LIN {X 0,Y 586.31,Z 664.399,A -85,B 0,C 180,E1 -9232.595,E2 -9232.595} C_VEL
LIN {X 0,Y 580.934,Z 684.929,A -85,B 0,C 180,E1 -9232.486,E2 -9232.486} C_VEL
LIN {X 0,Y 580.191,Z 691.532,A -85,B 0,C 180,E1 -9232.53,E2 -9232.53} C_VEL
LIN {X 0,Y 578.713,Z 743.986,A -85,B 0,C 180,E1 -9233.273,E2 -9233.273} C_VEL
LIN {X 0,Y 577.312,Z 767.92,A -85,B 0,C 180,E1 -9233.781,E2 -9233.781} C_VEL
LIN {X 0,Y 575.729,Z 789.042,A -85,B 0,C 180,E1 -9234.367,E2 -9234.367} C_VEL
LIN {X 0,Y 573.476,Z 813.615,A -85,B 0,C 180,E1 -9235.24,E2 -9235.24} C_VEL
LIN {X 0,Y 571.275,Z 833.863,A -85,B 0,C 180,E1 -9236.12,E2 -9236.12} C_VEL
LIN {X 0,Y 568.599,Z 856.085,A -85,B 0,C 180,E1 -9237.266,E2 -9237.266} C_VEL
LIN {X 0,Y 565.934,Z 875.723,A -85,B 0,C 180,E1 -9238.468,E2 -9238.468} C_VEL
LIN {X 0,Y 562.986,Z 896.638,A -85,B 0,C 180,E1 -9239.944,E2 -9239.944} C_VEL
LIN {X 0,Y 560.079,Z 915.772,A -85,B 0,C 180,E1 -9241.532,E2 -9241.532} C_VEL
LIN {X 0,Y 557.469,Z 932.739,A -85,B 0,C 180,E1 -9243.128,E2 -9243.128} C_VEL
LIN {X 0,Y 554.693,Z 950.508,A -85,B 0,C 180,E1 -9245.055,E2 -9245.055} C_VEL
LIN {X 0,Y 552.453,Z 965.214,A -85,B 0,C 180,E1 -9246.874,E2 -9246.874} C_VEL
LIN {X 0,Y 550.12,Z 981.104,A -85,B 0,C 180,E1 -9249.13,E2 -9249.13} C_VEL
LIN {X 0,Y 548.462,Z 993.237,A -85,B 0,C 180,E1 -9251.118,E2 -9251.118} C_VEL
LIN {X 0,Y 546.884,Z 1006.084,A -85,B 0,C 180,E1 -9253.537,E2 -9253.537} C_VEL
LIN {X 0,Y 545.776,Z 1016.202,A -85,B 0,C 180,E1 -9255.789,E2 -9255.789} C_VEL
LIN {X 0,Y 544.95,Z 1025.658,A -85,B 0,C 180,E1 -9258.249,E2 -9258.249} C_VEL
LIN {X 0,Y 544.408,Z 1033.231,A -85,B 0,C 180,E1 -9260.699,E2 -9260.699} C_VEL
LIN {X 0,Y 544.119,Z 1039.11,A -85,B 0,C 180,E1 -9263.034,E2 -9263.034} C_VEL
LIN {X 0,Y 543.975,Z 1043.859,A -85,B 0,C 180,E1 -9265.572,E2 -9265.572} C_VEL
LIN {X 0,Y 543.935,Z 1046.719,A -85,B 0,C 180,E1 -9267.788,E2 -9267.788} C_VEL
LIN {X 0,Y 543.91,Z 1048.63,A -85,B 0,C 180,E1 -9270.316,E2 -9270.316} C_VEL
LIN {X 0,Y 543.904,Z 1048.85,A -85,B 0,C 180,E1 -9272.74,E2 -9272.74} C_VEL
LIN {X 0,Y 543.911,Z 1047.945,A -85,B 0,C 180,E1 -9274.875,E2 -9274.875} C_VEL
LIN {X 0,Y 543.943,Z 1045.533,A -85,B 0,C 180,E1 -9277.393,E2 -9277.393} C_VEL
LIN {X 0,Y 544.029,Z 1041.559,A -85,B 0,C 180,E1 -9279.842,E2 -9279.842} C_VEL
LIN {X 0,Y 544.229,Z 1036.691,A -85,B 0,C 180,E1 -9282.09,E2 -9282.09} C_VEL
LIN {X 0,Y 544.667,Z 1029.45,A -85,B 0,C 180,E1 -9284.675,E2 -9284.675} C_VEL
LIN {X 0,Y 545.249,Z 1021.983,A -85,B 0,C 180,E1 -9286.843,E2 -9286.843} C_VEL
LIN {X 0,Y 546.21,Z 1012.263,A -85,B 0,C 180,E1 -9289.239,E2 -9289.239} C_VEL
LIN {X 0,Y 547.47,Z 1001.093,A -85,B 0,C 180,E1 -9291.537,E2 -9291.537} C_VEL
LIN {X 0,Y 549.156,Z 988.247,A -85,B 0,C 180,E1 -9293.842,E2 -9293.842} C_VEL
LIN {X 0,Y 551.198,Z 973.856,A -85,B 0,C 180,E1 -9296.04,E2 -9296.04} C_VEL
LIN {X 0,Y 553.43,Z 959.175,A -85,B 0,C 180,E1 -9298.018,E2 -9298.018} C_VEL
LIN {X 0,Y 556.081,Z 942.25,A -85,B 0,C 180,E1 -9299.992,E2 -9299.992} C_VEL
LIN {X 0,Y 558.6,Z 926.284,A -85,B 0,C 180,E1 -9301.632,E2 -9301.632} C_VEL
LIN {X 0,Y 561.851,Z 905.525,A -85,B 0,C 180,E1 -9303.483,E2 -9303.483} C_VEL
LIN {X 0,Y 564.509,Z 887.997,A -85,B 0,C 180,E1 -9304.836,E2 -9304.836} C_VEL
LIN {X 0,Y 567.634,Z 866.271,A -85,B 0,C 180,E1 -9306.289,E2 -9306.289} C_VEL
LIN {X 0,Y 570.163,Z 846.787,A -85,B 0,C 180,E1 -9307.399,E2 -9307.399} C_VEL
LIN {X 0,Y 572.736,Z 825.719,A -85,B 0,C 180,E1 -9308.426,E2 -9308.426} C_VEL
LIN {X 0,Y 575.102,Z 802.41,A -85,B 0,C 180,E1 -9309.358,E2 -9309.358} C_VEL
LIN {X 0,Y 577.063,Z 780.294,A -85,B 0,C 180,E1 -9310.073,E2 -9310.073} C_VEL
LIN {X 0,Y 578.78,Z 755.543,A -85,B 0,C 180,E1 -9310.679,E2 -9310.679} C_VEL
LIN {X 0,Y 579.816,Z 733.707,A -85,B 0,C 180,E1 -9311.068,E2 -9311.068} C_VEL
LIN {X 0,Y 586.618,Z 484.146,A -85,B 0,C 180,E1 -9314.52,E2 -9314.52} C_VEL
LIN {X 0,Y 588.402,Z 417.526,A -85,B 0,C 180,E1 -9315.46,E2 -9315.46} C_VEL
LIN {X 0,Y 575.019,Z 395.806,A -85,B 0,C 180,E1 -9317.164,E2 -9317.164} C_VEL
LIN {X 0,Y 561.085,Z 375.029,A -85,B 0,C 180,E1 -9319.053,E2 -9319.053} C_VEL
LIN {X 0,Y 553.737,Z 365.162,A -85,B 0,C 180,E1 -9320.097,E2 -9320.097} C_VEL
LIN {X 0,Y 550.099,Z 360.585,A -85,B 0,C 180,E1 -9320.627,E2 -9320.627} C_VEL
LIN {X 0,Y 549.271,Z 359.092,A -85,B 0,C 180,E1 -9320.758,E2 -9320.758} C_VEL
LIN {X 0,Y 546.699,Z 356.549,A -85,B 0,C 180,E1 -9321.129,E2 -9321.129} C_VEL
LIN {X 0,Y 545.557,Z 353.379,A -85,B 0,C 180,E1 -9321.337,E2 -9321.337} C_VEL
LIN {X 0,Y 545.5,Z 353.228,A -85,B 0,C 180,E1 -9324.654,E2 -9324.654} C_VEL
LIN {X 0,Y 545.56,Z 353.263,A -85,B 0,C 180,E1 -9327.893,E2 -9327.893} C_VEL
LIN {X 0,Y 545.51,Z 353.27,A -85,B 0,C 180,E1 -9331.06,E2 -9331.06} C_VEL
LIN {X 0,Y 545.517,Z 353.264,A -85,B 0,C 180,E1 -9334.486,E2 -9334.486} C_VEL
LIN {X 0,Y 545.558,Z 353.262,A -85,B 0,C 180,E1 -9337.752,E2 -9337.752} C_VEL
LIN {X 0,Y 545.507,Z 353.276,A -85,B 0,C 180,E1 -9341.051,E2 -9341.051} C_VEL
LIN {X 0,Y 545.541,Z 353.274,A -85,B 0,C 180,E1 -9344.37,E2 -9344.37} C_VEL
LIN {X 0,Y 545.517,Z 353.274,A -85,B 0,C 180,E1 -9347.509,E2 -9347.509} C_VEL
LIN {X 0,Y 545.506,Z 353.269,A -85,B 0,C 180,E1 -9350.93,E2 -9350.93} C_VEL
LIN {X 0,Y 545.561,Z 353.256,A -85,B 0,C 180,E1 -9354.109,E2 -9354.109} C_VEL
LIN {X 0,Y 545.504,Z 353.277,A -85,B 0,C 180,E1 -9357.394,E2 -9357.394} C_VEL
LIN {X 0,Y 545.533,Z 353.276,A -85,B 0,C 180,E1 -9360.735,E2 -9360.735} C_VEL
LIN {X 0,Y 545.532,Z 353.266,A -85,B 0,C 180,E1 -9363.994,E2 -9363.994} C_VEL
LIN {X 0,Y 545.502,Z 353.258,A -85,B 0,C 180,E1 -9367.266,E2 -9367.266} C_VEL
LIN {X 0,Y 545.559,Z 353.259,A -85,B 0,C 180,E1 -9370.454,E2 -9370.454} C_VEL
LIN {X 0,Y 545.504,Z 353.279,A -85,B 0,C 180,E1 -9373.719,E2 -9373.719} C_VEL
LIN {X 0,Y 545.528,Z 353.275,A -85,B 0,C 180,E1 -9377.053,E2 -9377.053} C_VEL
LIN {X 0,Y 545.531,Z 353.26,A -85,B 0,C 180,E1 -9380.268,E2 -9380.268} C_VEL
LIN {X 0,Y 545.502,Z 353.26,A -85,B 0,C 180,E1 -9383.553,E2 -9383.553} C_VEL
LIN {X 0,Y 545.562,Z 353.256,A -85,B 0,C 180,E1 -9386.803,E2 -9386.803} C_VEL
LIN {X 0,Y 545.503,Z 353.277,A -85,B 0,C 180,E1 -9389.905,E2 -9389.905} C_VEL
LIN {X 0,Y 545.538,Z 353.275,A -85,B 0,C 180,E1 -9393.232,E2 -9393.232} C_VEL
LIN {X 0,Y 545.522,Z 353.277,A -85,B 0,C 180,E1 -9396.432,E2 -9396.432} C_VEL
LIN {X 0,Y 545.547,Z 353.434,A -85,B 0,C 180,E1 -9398.499,E2 -9398.499} C_VEL
LIN {X 0,Y 546.943,Z 356.866,A -85,B 0,C 180,E1 -9399.103,E2 -9399.103} C_VEL
LIN {X 0,Y 552.731,Z 369.791,A -85,B 0,C 180,E1 -9401.346,E2 -9401.346} C_VEL
LIN {X 0,Y 553.923,Z 372.421,A -85,B 0,C 180,E1 -9401.731,E2 -9401.731} C_VEL
LIN {X 0,Y 566.29,Z 390.72,A -85,B 0,C 180,E1 -9403.483,E2 -9403.483} C_VEL
LIN {X 0,Y 578.478,Z 410.325,A -85,B 0,C 180,E1 -9405.11,E2 -9405.11} C_VEL
LIN {X 0,Y 588.478,Z 427.51,A -85,B 0,C 180,E1 -9406.38,E2 -9406.38} C_VEL
LIN {X 0,Y 581.411,Z 686.07,A -85,B 0,C 180,E1 -9409.961,E2 -9409.961} C_VEL
LIN {X 0,Y 579.185,Z 765.672,A -85,B 0,C 180,E1 -9411.076,E2 -9411.076} C_VEL
LIN {X 0,Y 577.58,Z 791.315,A -85,B 0,C 180,E1 -9411.595,E2 -9411.595} C_VEL
LIN {X 0,Y 575.8,Z 813.335,A -85,B 0,C 180,E1 -9412.197,E2 -9412.197} C_VEL
LIN {X 0,Y 573.376,Z 838.25,A -85,B 0,C 180,E1 -9413.076,E2 -9413.076} C_VEL
LIN {X 0,Y 571.195,Z 857.607,A -85,B 0,C 180,E1 -9413.91,E2 -9413.91} C_VEL
LIN {X 0,Y 568.389,Z 880.253,A -85,B 0,C 180,E1 -9415.062,E2 -9415.062} C_VEL
LIN {X 0,Y 565.532,Z 900.948,A -85,B 0,C 180,E1 -9416.322,E2 -9416.322} C_VEL
LIN {X 0,Y 562.652,Z 920.988,A -85,B 0,C 180,E1 -9417.723,E2 -9417.723} C_VEL
LIN {X 0,Y 559.666,Z 940.68,A -85,B 0,C 180,E1 -9419.332,E2 -9419.332} C_VEL
LIN {X 0,Y 557.039,Z 958.054,A -85,B 0,C 180,E1 -9420.947,E2 -9420.947} C_VEL
LIN {X 0,Y 554.171,Z 976.838,A -85,B 0,C 180,E1 -9422.955,E2 -9422.955} C_VEL
LIN {X 0,Y 551.96,Z 991.974,A -85,B 0,C 180,E1 -9424.804,E2 -9424.804} C_VEL
LIN {X 0,Y 549.686,Z 1008.315,A -85,B 0,C 180,E1 -9427.091,E2 -9427.091} C_VEL
LIN {X 0,Y 548.05,Z 1021.164,A -85,B 0,C 180,E1 -9429.159,E2 -9429.159} C_VEL
LIN {X 0,Y 546.494,Z 1034.945,A -85,B 0,C 180,E1 -9431.73,E2 -9431.73} C_VEL
LIN {X 0,Y 545.565,Z 1044.534,A -85,B 0,C 180,E1 -9433.825,E2 -9433.825} C_VEL
LIN {X 0,Y 544.805,Z 1054.257,A -85,B 0,C 180,E1 -9436.305,E2 -9436.305} C_VEL
LIN {X 0,Y 544.338,Z 1061.76,A -85,B 0,C 180,E1 -9438.665,E2 -9438.665} C_VEL
LIN {X 0,Y 544.07,Z 1067.856,A -85,B 0,C 180,E1 -9441.013,E2 -9441.013} C_VEL
LIN {X 0,Y 543.949,Z 1072.766,A -85,B 0,C 180,E1 -9443.562,E2 -9443.562} C_VEL
LIN {X 0,Y 543.918,Z 1075.604,A -85,B 0,C 180,E1 -9445.677,E2 -9445.677} C_VEL
LIN {X 0,Y 543.91,Z 1077.486,A -85,B 0,C 180,E1 -9447.998,E2 -9447.998} C_VEL
LIN {X 0,Y 543.902,Z 1077.918,A -85,B 0,C 180,E1 -9450.527,E2 -9450.527} C_VEL
LIN {X 0,Y 543.912,Z 1077.003,A -85,B 0,C 180,E1 -9452.74,E2 -9452.74} C_VEL
LIN {X 0,Y 543.934,Z 1074.679,A -85,B 0,C 180,E1 -9455.168,E2 -9455.168} C_VEL
LIN {X 0,Y 543.986,Z 1070.71,A -85,B 0,C 180,E1 -9457.605,E2 -9457.605} C_VEL
LIN {X 0,Y 544.145,Z 1066.055,A -85,B 0,C 180,E1 -9459.733,E2 -9459.733} C_VEL
LIN {X 0,Y 544.484,Z 1059.287,A -85,B 0,C 180,E1 -9462.192,E2 -9462.192} C_VEL
LIN {X 0,Y 545.031,Z 1051.054,A -85,B 0,C 180,E1 -9464.556,E2 -9464.556} C_VEL
LIN {X 0,Y 545.787,Z 1042.23,A -85,B 0,C 180,E1 -9466.716,E2 -9466.716} C_VEL
LIN {X 0,Y 547.007,Z 1030.206,A -85,B 0,C 180,E1 -9469.21,E2 -9469.21} C_VEL
LIN {X 0,Y 548.367,Z 1018.548,A -85,B 0,C 180,E1 -9471.289,E2 -9471.289} C_VEL
LIN {X 0,Y 550.294,Z 1003.93,A -85,B 0,C 180,E1 -9473.562,E2 -9473.562} C_VEL
LIN {X 0,Y 552.309,Z 989.361,A -85,B 0,C 180,E1 -9475.523,E2 -9475.523} C_VEL
LIN {X 0,Y 554.838,Z 972.333,A -85,B 0,C 180,E1 -9477.544,E2 -9477.544} C_VEL
LIN {X 0,Y 557.462,Z 954.481,A -85,B 0,C 180,E1 -9479.372,E2 -9479.372} C_VEL
LIN {X 0,Y 560.362,Z 935.264,A -85,B 0,C 180,E1 -9481.103,E2 -9481.103} C_VEL
LIN {X 0,Y 563.173,Z 915.778,A -85,B 0,C 180,E1 -9482.605,E2 -9482.605} C_VEL
LIN {X 0,Y 565.83,Z 896.882,A -85,B 0,C 180,E1 -9483.885,E2 -9483.885} C_VEL
LIN {X 0,Y 568.774,Z 873.901,A -85,B 0,C 180,E1 -9485.213,E2 -9485.213} C_VEL
LIN {X 0,Y 571.274,Z 853.014,A -85,B 0,C 180,E1 -9486.23,E2 -9486.23} C_VEL
LIN {X 0,Y 573.845,Z 828.285,A -85,B 0,C 180,E1 -9487.222,E2 -9487.222} C_VEL
LIN {X 0,Y 575.738,Z 807.183,A -85,B 0,C 180,E1 -9487.902,E2 -9487.902} C_VEL
LIN {X 0,Y 577.644,Z 781.289,A -85,B 0,C 180,E1 -9488.542,E2 -9488.542} C_VEL
LIN {X 0,Y 578.728,Z 759.201,A -85,B 0,C 180,E1 -9488.935,E2 -9488.935} C_VEL
LIN {X 0,Y 584.808,Z 519.513,A -85,B 0,C 180,E1 -9492.223,E2 -9492.223} C_VEL
LIN {X 0,Y 587.154,Z 426.916,A -85,B 0,C 180,E1 -9493.511,E2 -9493.511} C_VEL
LIN {X 0,Y 571.809,Z 400.651,A -85,B 0,C 180,E1 -9495.388,E2 -9495.388} C_VEL
LIN {X 0,Y 559.047,Z 380.64,A -85,B 0,C 180,E1 -9497.043,E2 -9497.043} C_VEL
LIN {X 0,Y 553.395,Z 371.842,A -85,B 0,C 180,E1 -9497.837,E2 -9497.837} C_VEL
LIN {X 0,Y 548.431,Z 360.447,A -85,B 0,C 180,E1 -9499.667,E2 -9499.667} C_VEL
LIN {X 0,Y 545.613,Z 353.686,A -85,B 0,C 180,E1 -9500.784,E2 -9500.784} C_VEL
LIN {X 0,Y 545.563,Z 353.268,A -85,B 0,C 180,E1 -9500.915,E2 -9500.915} C_VEL
LIN {X 0,Y 545.503,Z 353.282,A -85,B 0,C 180,E1 -9504.217,E2 -9504.217} C_VEL
LIN {X 0,Y 545.533,Z 353.276,A -85,B 0,C 180,E1 -9507.518,E2 -9507.518} C_VEL
LIN {X 0,Y 545.517,Z 353.275,A -85,B 0,C 180,E1 -9510.579,E2 -9510.579} C_VEL
LIN {X 0,Y 545.507,Z 353.274,A -85,B 0,C 180,E1 -9514.019,E2 -9514.019} C_VEL
LIN {X 0,Y 545.567,Z 353.251,A -85,B 0,C 180,E1 -9517.25,E2 -9517.25} C_VEL
LIN {X 0,Y 545.502,Z 353.261,A -85,B 0,C 180,E1 -9520.512,E2 -9520.512} C_VEL
LIN {X 0,Y 545.531,Z 353.274,A -85,B 0,C 180,E1 -9523.827,E2 -9523.827} C_VEL
LIN {X 0,Y 545.522,Z 353.268,A -85,B 0,C 180,E1 -9526.971,E2 -9526.971} C_VEL
LIN {X 0,Y 545.505,Z 353.253,A -85,B 0,C 180,E1 -9530.292,E2 -9530.292} C_VEL
LIN {X 0,Y 545.571,Z 353.272,A -85,B 0,C 180,E1 -9533.581,E2 -9533.581} C_VEL
LIN {X 0,Y 545.505,Z 353.27,A -85,B 0,C 180,E1 -9536.848,E2 -9536.848} C_VEL
LIN {X 0,Y 545.521,Z 353.252,A -85,B 0,C 180,E1 -9540.21,E2 -9540.21} C_VEL
LIN {X 0,Y 545.534,Z 353.275,A -85,B 0,C 180,E1 -9543.362,E2 -9543.362} C_VEL
LIN {X 0,Y 545.504,Z 353.259,A -85,B 0,C 180,E1 -9546.631,E2 -9546.631} C_VEL
LIN {X 0,Y 545.561,Z 353.262,A -85,B 0,C 180,E1 -9549.814,E2 -9549.814} C_VEL
LIN {X 0,Y 545.509,Z 353.276,A -85,B 0,C 180,E1 -9553.137,E2 -9553.137} C_VEL
LIN {X 0,Y 545.519,Z 353.257,A -85,B 0,C 180,E1 -9556.541,E2 -9556.541} C_VEL
LIN {X 0,Y 545.545,Z 353.267,A -85,B 0,C 180,E1 -9559.709,E2 -9559.709} C_VEL
LIN {X 0,Y 545.508,Z 353.279,A -85,B 0,C 180,E1 -9562.981,E2 -9562.981} C_VEL
LIN {X 0,Y 545.562,Z 353.255,A -85,B 0,C 180,E1 -9566.212,E2 -9566.212} C_VEL
LIN {X 0,Y 545.51,Z 353.258,A -85,B 0,C 180,E1 -9569.422,E2 -9569.422} C_VEL
LIN {X 0,Y 545.518,Z 353.261,A -85,B 0,C 180,E1 -9572.857,E2 -9572.857} C_VEL
LIN {X 0,Y 545.552,Z 353.265,A -85,B 0,C 180,E1 -9576.073,E2 -9576.073} C_VEL
LIN {X 0,Y 545.505,Z 353.271,A -85,B 0,C 180,E1 -9579.361,E2 -9579.361} C_VEL
LIN {X 0,Y 545.556,Z 353.244,A -85,B 0,C 180,E1 -9582.555,E2 -9582.555} C_VEL
LIN {X 0,Y 545.524,Z 353.391,A -85,B 0,C 180,E1 -9583.36,E2 -9583.36} C_VEL
LIN {X 0,Y 546.695,Z 356.539,A -85,B 0,C 180,E1 -9583.556,E2 -9583.556} C_VEL
LIN {X 0,Y 549.535,Z 359.67,A -85,B 0,C 180,E1 -9583.941,E2 -9583.941} C_VEL
LIN {X 0,Y 552.166,Z 363.52,A -85,B 0,C 180,E1 -9584.31,E2 -9584.31} C_VEL
LIN {X 0,Y 562.945,Z 378.525,A -85,B 0,C 180,E1 -9585.746,E2 -9585.746} C_VEL
LIN {X 0,Y 577.16,Z 400.506,A -85,B 0,C 180,E1 -9587.545,E2 -9587.545} C_VEL
LIN {X 0,Y 587.285,Z 417.698,A -85,B 0,C 180,E1 -9588.768,E2 -9588.768} C_VEL
LIN {X 0,Y 580.842,Z 665.424,A -85,B 0,C 180,E1 -9592.174,E2 -9592.174} C_VEL
LIN {X 0,Y 580.191,Z 691.532,A -85,B 0,C 180,E1 -9592.53,E2 -9592.53} C_VEL
LIN {X 0,Y 579.237,Z 699.223,A -85,B 0,C 180,E1 -9592.574,E2 -9592.574} C_VEL
LIN {X 0,Y 573.858,Z 719.75,A -85,B 0,C 180,E1 -9592.463,E2 -9592.463} C_VEL
LIN {X 0,Y 573.08,Z 726.354,A -85,B 0,C 180,E1 -9592.505,E2 -9592.505} C_VEL
LIN {X 0,Y 572.003,Z 751.824,A -85,B 0,C 180,E1 -9592.929,E2 -9592.929} C_VEL
LIN {X 0,Y 570.686,Z 772.366,A -85,B 0,C 180,E1 -9593.398,E2 -9593.398} C_VEL
LIN {X 0,Y 568.636,Z 797.064,A -85,B 0,C 180,E1 -9594.137,E2 -9594.137} C_VEL
LIN {X 0,Y 566.572,Z 817.66,A -85,B 0,C 180,E1 -9594.917,E2 -9594.917} C_VEL
LIN {X 0,Y 564.003,Z 840.035,A -85,B 0,C 180,E1 -9595.929,E2 -9595.929} C_VEL
LIN {X 0,Y 561.11,Z 861.963,A -85,B 0,C 180,E1 -9597.138,E2 -9597.138} C_VEL
LIN {X 0,Y 558.208,Z 882.64,A -85,B 0,C 180,E1 -9598.463,E2 -9598.463} C_VEL
LIN {X 0,Y 555.065,Z 903.039,A -85,B 0,C 180,E1 -9600.008,E2 -9600.008} C_VEL
LIN {X 0,Y 552.221,Z 921.02,A -85,B 0,C 180,E1 -9601.562,E2 -9601.562} C_VEL
LIN {X 0,Y 549.207,Z 939.328,A -85,B 0,C 180,E1 -9603.393,E2 -9603.393} C_VEL
LIN {X 0,Y 546.755,Z 954.528,A -85,B 0,C 180,E1 -9605.126,E2 -9605.126} C_VEL
LIN {X 0,Y 543.979,Z 971.939,A -85,B 0,C 180,E1 -9607.408,E2 -9607.408} C_VEL
LIN {X 0,Y 542.016,Z 984.923,A -85,B 0,C 180,E1 -9609.369,E2 -9609.369} C_VEL
LIN {X 0,Y 539.993,Z 999.294,A -85,B 0,C 180,E1 -9611.876,E2 -9611.876} C_VEL
LIN {X 0,Y 538.655,Z 1010.001,A -85,B 0,C 180,E1 -9614.061,E2 -9614.061} C_VEL
LIN {X 0,Y 537.499,Z 1020.862,A -85,B 0,C 180,E1 -9616.663,E2 -9616.663} C_VEL
LIN {X 0,Y 536.808,Z 1028.736,A -85,B 0,C 180,E1 -9618.939,E2 -9618.939} C_VEL
LIN {X 0,Y 536.338,Z 1035.901,A -85,B 0,C 180,E1 -9621.423,E2 -9621.423} C_VEL
LIN {X 0,Y 536.068,Z 1041.325,A -85,B 0,C 180,E1 -9623.897,E2 -9623.897} C_VEL
LIN {X 0,Y 535.965,Z 1045.057,A -85,B 0,C 180,E1 -9626.149,E2 -9626.149} C_VEL
LIN {X 0,Y 535.926,Z 1047.938,A -85,B 0,C 180,E1 -9628.824,E2 -9628.824} C_VEL
LIN {X 0,Y 535.915,Z 1049.006,A -85,B 0,C 180,E1 -9631.069,E2 -9631.069} C_VEL
LIN {X 0,Y 535.915,Z 1048.946,A -85,B 0,C 180,E1 -9633.316,E2 -9633.316} C_VEL
LIN {X 0,Y 535.937,Z 1047.259,A -85,B 0,C 180,E1 -9636.057,E2 -9636.057} C_VEL
LIN {X 0,Y 535.982,Z 1044.441,A -85,B 0,C 180,E1 -9638.367,E2 -9638.367} C_VEL
LIN {X 0,Y 536.119,Z 1040.085,A -85,B 0,C 180,E1 -9640.858,E2 -9640.858} C_VEL
LIN {X 0,Y 536.43,Z 1034.004,A -85,B 0,C 180,E1 -9643.364,E2 -9643.364} C_VEL
LIN {X 0,Y 536.937,Z 1027.114,A -85,B 0,C 180,E1 -9645.665,E2 -9645.665} C_VEL
LIN {X 0,Y 537.836,Z 1017.399,A -85,B 0,C 180,E1 -9648.312,E2 -9648.312} C_VEL
LIN {X 0,Y 538.943,Z 1007.721,A -85,B 0,C 180,E1 -9650.527,E2 -9650.527} C_VEL
LIN {X 0,Y 540.651,Z 994.638,A -85,B 0,C 180,E1 -9653.084,E2 -9653.084} C_VEL
LIN {X 0,Y 542.438,Z 982.245,A -85,B 0,C 180,E1 -9655.166,E2 -9655.166} C_VEL
LIN {X 0,Y 544.874,Z 966.806,A -85,B 0,C 180,E1 -9657.426,E2 -9657.426} C_VEL
LIN {X 0,Y 547.286,Z 951.914,A -85,B 0,C 180,E1 -9659.317,E2 -9659.317} C_VEL
LIN {X 0,Y 550.212,Z 934.606,A -85,B 0,C 180,E1 -9661.254,E2 -9661.254} C_VEL
LIN {X 0,Y 553.189,Z 916.48,A -85,B 0,C 180,E1 -9662.998,E2 -9662.998} C_VEL
LIN {X 0,Y 556.389,Z 896.896,A -85,B 0,C 180,E1 -9664.654,E2 -9664.654} C_VEL
LIN {X 0,Y 559.532,Z 876.209,A -85,B 0,C 180,E1 -9666.137,E2 -9666.137} C_VEL
LIN {X 0,Y 562.581,Z 855.295,A -85,B 0,C 180,E1 -9667.434,E2 -9667.434} C_VEL
LIN {X 0,Y 565.399,Z 833.348,A -85,B 0,C 180,E1 -9668.57,E2 -9668.57} C_VEL
LIN {X 0,Y 567.648,Z 814.001,A -85,B 0,C 180,E1 -9669.421,E2 -9669.421} C_VEL
LIN {X 0,Y 570.061,Z 789.555,A -85,B 0,C 180,E1 -9670.301,E2 -9670.301} C_VEL
LIN {X 0,Y 571.773,Z 768.263,A -85,B 0,C 180,E1 -9670.9,E2 -9670.9} C_VEL
LIN {X 0,Y 573.277,Z 744.413,A -85,B 0,C 180,E1 -9671.413,E2 -9671.413} C_VEL
LIN {X 0,Y 574.895,Z 692.081,A -85,B 0,C 180,E1 -9672.167,E2 -9672.167} C_VEL
LIN {X 0,Y 582.054,Z 442.595,A -85,B 0,C 180,E1 -9675.648,E2 -9675.648} C_VEL
LIN {X 0,Y 582.588,Z 420.937,A -85,B 0,C 180,E1 -9675.965,E2 -9675.965} C_VEL
LIN {X 0,Y 570.546,Z 401.354,A -85,B 0,C 180,E1 -9677.533,E2 -9677.533} C_VEL
LIN {X 0,Y 557.188,Z 381.281,A -85,B 0,C 180,E1 -9679.382,E2 -9679.382} C_VEL
LIN {X 0,Y 548.562,Z 369.951,A -85,B 0,C 180,E1 -9680.63,E2 -9680.63} C_VEL
LIN {X 0,Y 545.139,Z 365.328,A -85,B 0,C 180,E1 -9681.149,E2 -9681.149} C_VEL
LIN {X 0,Y 542.298,Z 361.709,A -85,B 0,C 180,E1 -9681.584,E2 -9681.584} C_VEL
LIN {X 0,Y 541.197,Z 359.978,A -85,B 0,C 180,E1 -9681.762,E2 -9681.762} C_VEL
LIN {X 0,Y 538.622,Z 357.309,A -85,B 0,C 180,E1 -9682.154,E2 -9682.154} C_VEL
LIN {X 0,Y 537.573,Z 354.248,A -85,B 0,C 180,E1 -9682.371,E2 -9682.371} C_VEL
LIN {X 0,Y 537.62,Z 354.227,A -85,B 0,C 180,E1 -9685.699,E2 -9685.699} C_VEL
LIN {X 0,Y 537.569,Z 354.256,A -85,B 0,C 180,E1 -9688.987,E2 -9688.987} C_VEL
LIN {X 0,Y 537.581,Z 354.261,A -85,B 0,C 180,E1 -9692.41,E2 -9692.41} C_VEL
LIN {X 0,Y 537.617,Z 354.253,A -85,B 0,C 180,E1 -9695.73,E2 -9695.73} C_VEL
LIN {X 0,Y 537.566,Z 354.256,A -85,B 0,C 180,E1 -9699.025,E2 -9699.025} C_VEL
LIN {X 0,Y 537.599,Z 354.249,A -85,B 0,C 180,E1 -9702.352,E2 -9702.352} C_VEL
LIN {X 0,Y 537.575,Z 354.255,A -85,B 0,C 180,E1 -9705.457,E2 -9705.457} C_VEL
LIN {X 0,Y 537.571,Z 354.263,A -85,B 0,C 180,E1 -9708.846,E2 -9708.846} C_VEL
LIN {X 0,Y 537.632,Z 354.263,A -85,B 0,C 180,E1 -9712.197,E2 -9712.197} C_VEL
LIN {X 0,Y 537.571,Z 354.259,A -85,B 0,C 180,E1 -9715.537,E2 -9715.537} C_VEL
LIN {X 0,Y 537.568,Z 354.251,A -85,B 0,C 180,E1 -9719.041,E2 -9719.041} C_VEL
LIN {X 0,Y 537.619,Z 354.246,A -85,B 0,C 180,E1 -9722.238,E2 -9722.238} C_VEL
LIN {X 0,Y 537.566,Z 354.269,A -85,B 0,C 180,E1 -9725.55,E2 -9725.55} C_VEL
LIN {X 0,Y 537.592,Z 354.266,A -85,B 0,C 180,E1 -9728.881,E2 -9728.881} C_VEL
LIN {X 0,Y 537.593,Z 354.248,A -85,B 0,C 180,E1 -9732.133,E2 -9732.133} C_VEL
LIN {X 0,Y 537.562,Z 354.246,A -85,B 0,C 180,E1 -9735.426,E2 -9735.426} C_VEL
LIN {X 0,Y 537.623,Z 354.245,A -85,B 0,C 180,E1 -9738.656,E2 -9738.656} C_VEL
LIN {X 0,Y 537.569,Z 354.267,A -85,B 0,C 180,E1 -9741.954,E2 -9741.954} C_VEL
LIN {X 0,Y 537.571,Z 354.267,A -85,B 0,C 180,E1 -9745.446,E2 -9745.446} C_VEL
LIN {X 0,Y 537.636,Z 354.264,A -85,B 0,C 180,E1 -9748.796,E2 -9748.796} C_VEL
LIN {X 0,Y 537.566,Z 354.269,A -85,B 0,C 180,E1 -9752.013,E2 -9752.013} C_VEL
LIN {X 0,Y 537.581,Z 354.27,A -85,B 0,C 180,E1 -9755.445,E2 -9755.445} C_VEL
LIN {X 0,Y 537.598,Z 354.432,A -85,B 0,C 180,E1 -9757.558,E2 -9757.558} C_VEL
LIN {X 0,Y 538.888,Z 357.777,A -85,B 0,C 180,E1 -9758.161,E2 -9758.161} C_VEL
LIN {X 0,Y 541.452,Z 363.112,A -85,B 0,C 180,E1 -9759.166,E2 -9759.166} C_VEL
LIN {X 0,Y 545.365,Z 371.859,A -85,B 0,C 180,E1 -9760.677,E2 -9760.677} C_VEL
LIN {X 0,Y 558.222,Z 390.685,A -85,B 0,C 180,E1 -9762.581,E2 -9762.581} C_VEL
LIN {X 0,Y 572.345,Z 413.012,A -85,B 0,C 180,E1 -9764.529,E2 -9764.529} C_VEL
LIN {X 0,Y 582.655,Z 430.956,A -85,B 0,C 180,E1 -9765.879,E2 -9765.879} C_VEL
LIN {X 0,Y 575.261,Z 689.165,A -85,B 0,C 180,E1 -9769.484,E2 -9769.484} C_VEL
LIN {X 0,Y 573.021,Z 765.526,A -85,B 0,C 180,E1 -9770.564,E2 -9770.564} C_VEL
LIN {X 0,Y 571.362,Z 791.034,A -85,B 0,C 180,E1 -9771.083,E2 -9771.083} C_VEL
LIN {X 0,Y 569.508,Z 813.006,A -85,B 0,C 180,E1 -9771.687,E2 -9771.687} C_VEL
LIN {X 0,Y 567.08,Z 837.01,A -85,B 0,C 180,E1 -9772.532,E2 -9772.532} C_VEL
LIN {X 0,Y 564.664,Z 857.615,A -85,B 0,C 180,E1 -9773.426,E2 -9773.426} C_VEL
LIN {X 0,Y 561.706,Z 880.381,A -85,B 0,C 180,E1 -9774.596,E2 -9774.596} C_VEL
LIN {X 0,Y 558.718,Z 901.112,A -85,B 0,C 180,E1 -9775.872,E2 -9775.872} C_VEL
LIN {X 0,Y 555.626,Z 921.636,A -85,B 0,C 180,E1 -9777.325,E2 -9777.325} C_VEL
LIN {X 0,Y 552.492,Z 941.178,A -85,B 0,C 180,E1 -9778.95,E2 -9778.95} C_VEL
LIN {X 0,Y 549.706,Z 958.728,A -85,B 0,C 180,E1 -9780.608,E2 -9780.608} C_VEL
LIN {X 0,Y 546.81,Z 976.686,A -85,B 0,C 180,E1 -9782.561,E2 -9782.561} C_VEL
LIN {X 0,Y 544.466,Z 991.807,A -85,B 0,C 180,E1 -9784.433,E2 -9784.433} C_VEL
LIN {X 0,Y 542.061,Z 1008.127,A -85,B 0,C 180,E1 -9786.75,E2 -9786.75} C_VEL
LIN {X 0,Y 540.311,Z 1021.029,A -85,B 0,C 180,E1 -9788.859,E2 -9788.859} C_VEL
LIN {X 0,Y 538.643,Z 1034.899,A -85,B 0,C 180,E1 -9791.492,E2 -9791.492} C_VEL
LIN {X 0,Y 537.634,Z 1044.778,A -85,B 0,C 180,E1 -9793.69,E2 -9793.69} C_VEL
LIN {X 0,Y 536.807,Z 1054.754,A -85,B 0,C 180,E1 -9796.317,E2 -9796.317} C_VEL
LIN {X 0,Y 536.35,Z 1061.849,A -85,B 0,C 180,E1 -9798.603,E2 -9798.603} C_VEL
LIN {X 0,Y 536.065,Z 1068.155,A -85,B 0,C 180,E1 -9801.094,E2 -9801.094} C_VEL
LIN {X 0,Y 535.95,Z 1072.713,A -85,B 0,C 180,E1 -9803.573,E2 -9803.573} C_VEL
LIN {X 0,Y 535.918,Z 1075.505,A -85,B 0,C 180,E1 -9805.72,E2 -9805.72} C_VEL
LIN {X 0,Y 535.906,Z 1077.409,A -85,B 0,C 180,E1 -9808.182,E2 -9808.182} C_VEL
LIN {X 0,Y 535.906,Z 1077.682,A -85,B 0,C 180,E1 -9810.641,E2 -9810.641} C_VEL
LIN {X 0,Y 535.915,Z 1076.789,A -85,B 0,C 180,E1 -9812.78,E2 -9812.78} C_VEL
LIN {X 0,Y 535.934,Z 1074.466,A -85,B 0,C 180,E1 -9815.245,E2 -9815.245} C_VEL
LIN {X 0,Y 535.99,Z 1070.496,A -85,B 0,C 180,E1 -9817.719,E2 -9817.719} C_VEL
LIN {X 0,Y 536.155,Z 1065.839,A -85,B 0,C 180,E1 -9819.879,E2 -9819.879} C_VEL
LIN {X 0,Y 536.526,Z 1058.886,A -85,B 0,C 180,E1 -9822.432,E2 -9822.432} C_VEL
LIN {X 0,Y 537.135,Z 1050.426,A -85,B 0,C 180,E1 -9824.886,E2 -9824.886} C_VEL
LIN {X 0,Y 538.052,Z 1040.616,A -85,B 0,C 180,E1 -9827.298,E2 -9827.298} C_VEL
LIN {X 0,Y 539.349,Z 1028.823,A -85,B 0,C 180,E1 -9829.719,E2 -9829.719} C_VEL
LIN {X 0,Y 540.915,Z 1016.457,A -85,B 0,C 180,E1 -9831.925,E2 -9831.925} C_VEL
LIN {X 0,Y 543.014,Z 1001.327,A -85,B 0,C 180,E1 -9834.244,E2 -9834.244} C_VEL
LIN {X 0,Y 545.091,Z 987.372,A -85,B 0,C 180,E1 -9836.119,E2 -9836.119} C_VEL
LIN {X 0,Y 547.921,Z 969.064,A -85,B 0,C 180,E1 -9838.265,E2 -9838.265} C_VEL
LIN {X 0,Y 550.435,Z 952.988,A -85,B 0,C 180,E1 -9839.91,E2 -9839.91} C_VEL
LIN {X 0,Y 553.61,Z 932.836,A -85,B 0,C 180,E1 -9841.713,E2 -9841.713} C_VEL
LIN {X 0,Y 556.371,Z 914.575,A -85,B 0,C 180,E1 -9843.125,E2 -9843.125} C_VEL
LIN {X 0,Y 559.385,Z 894.047,A -85,B 0,C 180,E1 -9844.516,E2 -9844.516} C_VEL
LIN {X 0,Y 562.224,Z 872.47,A -85,B 0,C 180,E1 -9845.748,E2 -9845.748} C_VEL
LIN {X 0,Y 564.952,Z 850.686,A -85,B 0,C 180,E1 -9846.805,E2 -9846.805} C_VEL
LIN {X 0,Y 567.425,Z 827.51,A -85,B 0,C 180,E1 -9847.727,E2 -9847.727} C_VEL
LIN {X 0,Y 569.383,Z 806.505,A -85,B 0,C 180,E1 -9848.405,E2 -9848.405} C_VEL
LIN {X 0,Y 571.327,Z 780.86,A -85,B 0,C 180,E1 -9849.041,E2 -9849.041} C_VEL
LIN {X 0,Y 572.445,Z 758.816,A -85,B 0,C 180,E1 -9849.435,E2 -9849.435} C_VEL
LIN {X 0,Y 578.832,Z 518.494,A -85,B 0,C 180,E1 -9852.761,E2 -9852.761} C_VEL
LIN {X 0,Y 581.183,Z 430.246,A -85,B 0,C 180,E1 -9853.998,E2 -9853.998} C_VEL
LIN {X 0,Y 567.071,Z 405.931,A -85,B 0,C 180,E1 -9855.766,E2 -9855.766} C_VEL
LIN {X 0,Y 554.721,Z 386.396,A -85,B 0,C 180,E1 -9857.402,E2 -9857.402} C_VEL
LIN {X 0,Y 546.313,Z 373.784,A -85,B 0,C 180,E1 -9858.575,E2 -9858.575} C_VEL
LIN {X 0,Y 544.919,Z 371.558,A -85,B 0,C 180,E1 -9858.796,E2 -9858.796} C_VEL
LIN {X 0,Y 540.498,Z 361.439,A -85,B 0,C 180,E1 -9860.482,E2 -9860.482} C_VEL
LIN {X 0,Y 538.801,Z 357.546,A -85,B 0,C 180,E1 -9861.152,E2 -9861.152} C_VEL
LIN {X 0,Y 537.572,Z 354.265,A -85,B 0,C 180,E1 -9861.729,E2 -9861.729} C_VEL
LIN {X 0,Y 537.62,Z 354.251,A -85,B 0,C 180,E1 -9865.052,E2 -9865.052} C_VEL
LIN {X 0,Y 537.562,Z 354.258,A -85,B 0,C 180,E1 -9868.238,E2 -9868.238} C_VEL
LIN {X 0,Y 537.599,Z 354.255,A -85,B 0,C 180,E1 -9871.566,E2 -9871.566} C_VEL
LIN {X 0,Y 537.588,Z 354.264,A -85,B 0,C 180,E1 -9874.79,E2 -9874.79} C_VEL
LIN {X 0,Y 537.563,Z 354.266,A -85,B 0,C 180,E1 -9878.16,E2 -9878.16} C_VEL
LIN {X 0,Y 537.619,Z 354.241,A -85,B 0,C 180,E1 -9881.456,E2 -9881.456} C_VEL
LIN {X 0,Y 537.569,Z 354.256,A -85,B 0,C 180,E1 -9884.685,E2 -9884.685} C_VEL
LIN {X 0,Y 537.573,Z 354.267,A -85,B 0,C 180,E1 -9888.194,E2 -9888.194} C_VEL
LIN {X 0,Y 537.626,Z 354.242,A -85,B 0,C 180,E1 -9891.551,E2 -9891.551} C_VEL
LIN {X 0,Y 537.565,Z 354.251,A -85,B 0,C 180,E1 -9894.771,E2 -9894.771} C_VEL
LIN {X 0,Y 537.584,Z 354.268,A -85,B 0,C 180,E1 -9898.188,E2 -9898.188} C_VEL
LIN {X 0,Y 537.6,Z 354.237,A -85,B 0,C 180,E1 -9901.386,E2 -9901.386} C_VEL
LIN {X 0,Y 537.564,Z 354.258,A -85,B 0,C 180,E1 -9904.694,E2 -9904.694} C_VEL
LIN {X 0,Y 537.617,Z 354.259,A -85,B 0,C 180,E1 -9908.018,E2 -9908.018} C_VEL
LIN {X 0,Y 537.575,Z 354.238,A -85,B 0,C 180,E1 -9911.262,E2 -9911.262} C_VEL
LIN {X 0,Y 537.569,Z 354.259,A -85,B 0,C 180,E1 -9914.713,E2 -9914.713} C_VEL
LIN {X 0,Y 537.626,Z 354.257,A -85,B 0,C 180,E1 -9917.983,E2 -9917.983} C_VEL
LIN {X 0,Y 537.569,Z 354.245,A -85,B 0,C 180,E1 -9921.272,E2 -9921.272} C_VEL
LIN {X 0,Y 537.585,Z 354.247,A -85,B 0,C 180,E1 -9924.622,E2 -9924.622} C_VEL
LIN {X 0,Y 537.619,Z 354.263,A -85,B 0,C 180,E1 -9927.949,E2 -9927.949} C_VEL
LIN {X 0,Y 537.57,Z 354.269,A -85,B 0,C 180,E1 -9931.262,E2 -9931.262} C_VEL
LIN {X 0,Y 537.607,Z 354.258,A -85,B 0,C 180,E1 -9934.56,E2 -9934.56} C_VEL
LIN {X 0,Y 537.591,Z 354.263,A -85,B 0,C 180,E1 -9937.864,E2 -9937.864} C_VEL
LIN {X 0,Y 537.573,Z 354.271,A -85,B 0,C 180,E1 -9941.182,E2 -9941.182} C_VEL
LIN {X 0,Y 537.651,Z 354.44,A -85,B 0,C 180,E1 -9942.44,E2 -9942.44} C_VEL
LIN {X 0,Y 538.856,Z 357.626,A -85,B 0,C 180,E1 -9942.65,E2 -9942.65} C_VEL
LIN {X 0,Y 541.64,Z 360.745,A -85,B 0,C 180,E1 -9943.045,E2 -9943.045} C_VEL
LIN {X 0,Y 544.3,Z 364.596,A -85,B 0,C 180,E1 -9943.433,E2 -9943.433} C_VEL
LIN {X 0,Y 545.871,Z 366.544,A -85,B 0,C 180,E1 -9943.653,E2 -9943.653} C_VEL
LIN {X 0,Y 558.69,Z 384.425,A -85,B 0,C 180,E1 -9945.405,E2 -9945.405} C_VEL
LIN {X 0,Y 572.771,Z 406.422,A -85,B 0,C 180,E1 -9947.222,E2 -9947.222} C_VEL
LIN {X 0,Y 581.317,Z 421.073,A -85,B 0,C 180,E1 -9948.28,E2 -9948.28} C_VEL
LIN {X 0,Y 574.594,Z 667.992,A -85,B 0,C 180,E1 -9951.703,E2 -9951.703} C_VEL
LIN {X 0,Y 573.08,Z 726.354,A -85,B 0,C 180,E1 -9952.505,E2 -9952.505} C_VEL
LIN {X 0,Y 572.024,Z 734.039,A -85,B 0,C 180,E1 -9952.548,E2 -9952.548} C_VEL
LIN {X 0,Y 566.404,Z 753.361,A -85,B 0,C 180,E1 -9952.511,E2 -9952.511} C_VEL
LIN {X 0,Y 565.216,Z 760.968,A -85,B 0,C 180,E1 -9952.606,E2 -9952.606} C_VEL
LIN {X 0,Y 563.322,Z 785.096,A -85,B 0,C 180,E1 -9953.249,E2 -9953.249} C_VEL
LIN {X 0,Y 561.204,Z 807.81,A -85,B 0,C 180,E1 -9954.019,E2 -9954.019} C_VEL
LIN {X 0,Y 558.613,Z 830.665,A -85,B 0,C 180,E1 -9954.993,E2 -9954.993} C_VEL
LIN {X 0,Y 556.166,Z 849.641,A -85,B 0,C 180,E1 -9955.949,E2 -9955.949} C_VEL
LIN {X 0,Y 552.913,Z 872.771,A -85,B 0,C 180,E1 -9957.329,E2 -9957.329} C_VEL
LIN {X 0,Y 550.056,Z 891.211,A -85,B 0,C 180,E1 -9958.62,E2 -9958.62} C_VEL
LIN {X 0,Y 546.807,Z 911.299,A -85,B 0,C 180,E1 -9960.234,E2 -9960.234} C_VEL
LIN {X 0,Y 543.754,Z 929.256,A -85,B 0,C 180,E1 -9961.917,E2 -9961.917} C_VEL
LIN {X 0,Y 540.822,Z 946.72,A -85,B 0,C 180,E1 -9963.777,E2 -9963.777} C_VEL
LIN {X 0,Y 538.054,Z 962.697,A -85,B 0,C 180,E1 -9965.752,E2 -9965.752} C_VEL
LIN {X 0,Y 535.694,Z 977.225,A -85,B 0,C 180,E1 -9967.79,E2 -9967.79} C_VEL
LIN {X 0,Y 533.393,Z 991.816,A -85,B 0,C 180,E1 -9970.166,E2 -9970.166} C_VEL
LIN {X 0,Y 531.807,Z 1003.018,A -85,B 0,C 180,E1 -9972.267,E2 -9972.267} C_VEL
LIN {X 0,Y 530.282,Z 1015.096,A -85,B 0,C 180,E1 -9974.917,E2 -9974.917} C_VEL
LIN {X 0,Y 529.372,Z 1023.567,A -85,B 0,C 180,E1 -9977.122,E2 -9977.122} C_VEL
LIN {X 0,Y 528.655,Z 1032.053,A -85,B 0,C 180,E1 -9979.759,E2 -9979.759} C_VEL
LIN {X 0,Y 528.245,Z 1038.188,A -85,B 0,C 180,E1 -9982.167,E2 -9982.167} C_VEL
LIN {X 0,Y 528.036,Z 1043.216,A -85,B 0,C 180,E1 -9984.676,E2 -9984.676} C_VEL
LIN {X 0,Y 527.946,Z 1046.764,A -85,B 0,C 180,E1 -9987.286,E2 -9987.286} C_VEL
LIN {X 0,Y 527.918,Z 1048.638,A -85,B 0,C 180,E1 -9989.566,E2 -9989.566} C_VEL
LIN {X 0,Y 527.911,Z 1049.399,A -85,B 0,C 180,E1 -9992.171,E2 -9992.171} C_VEL
LIN {X 0,Y 527.915,Z 1048.551,A -85,B 0,C 180,E1 -9994.672,E2 -9994.672} C_VEL
LIN {X 0,Y 527.949,Z 1046.609,A -85,B 0,C 180,E1 -9996.962,E2 -9996.962} C_VEL
LIN {X 0,Y 528.045,Z 1042.69,A -85,B 0,C 180,E1 -9999.702,E2 -9999.702} C_VEL
LIN {X 0,Y 528.255,Z 1037.986,A -85,B 0,C 180,E1 -10002.017,E2 -10002.017} C_VEL
LIN {X 0,Y 528.707,Z 1031.428,A -85,B 0,C 180,E1 -10004.568,E2 -10004.568} C_VEL
LIN {X 0,Y 529.433,Z 1022.993,A -85,B 0,C 180,E1 -10007.135,E2 -10007.135} C_VEL
LIN {X 0,Y 530.503,Z 1013.389,A -85,B 0,C 180,E1 -10009.603,E2 -10009.603} C_VEL
LIN {X 0,Y 532.004,Z 1001.752,A -85,B 0,C 180,E1 -10012.091,E2 -10012.091} C_VEL
LIN {X 0,Y 533.792,Z 989.652,A -85,B 0,C 180,E1 -10014.337,E2 -10014.337} C_VEL
LIN {X 0,Y 536.05,Z 975.49,A -85,B 0,C 180,E1 -10016.594,E2 -10016.594} C_VEL
LIN {X 0,Y 538.508,Z 960.941,A -85,B 0,C 180,E1 -10018.623,E2 -10018.623} C_VEL
LIN {X 0,Y 541.584,Z 943.283,A -85,B 0,C 180,E1 -10020.758,E2 -10020.758} C_VEL
LIN {X 0,Y 544.361,Z 927.384,A -85,B 0,C 180,E1 -10022.436,E2 -10022.436} C_VEL
LIN {X 0,Y 547.94,Z 906.773,A -85,B 0,C 180,E1 -10024.324,E2 -10024.324} C_VEL
LIN {X 0,Y 550.833,Z 889.337,A -85,B 0,C 180,E1 -10025.704,E2 -10025.704} C_VEL
LIN {X 0,Y 554.113,Z 868.732,A -85,B 0,C 180,E1 -10027.128,E2 -10027.128} C_VEL
LIN {X 0,Y 557.021,Z 848.148,A -85,B 0,C 180,E1 -10028.33,E2 -10028.33} C_VEL
LIN {X 0,Y 559.753,Z 827.581,A -85,B 0,C 180,E1 -10029.356,E2 -10029.356} C_VEL
LIN {X 0,Y 562.402,Z 803.981,A -85,B 0,C 180,E1 -10030.327,E2 -10030.327} C_VEL
LIN {X 0,Y 564.454,Z 782.628,A -85,B 0,C 180,E1 -10031.036,E2 -10031.036} C_VEL
LIN {X 0,Y 566.444,Z 756.724,A -85,B 0,C 180,E1 -10031.692,E2 -10031.692} C_VEL
LIN {X 0,Y 567.573,Z 734.884,A -85,B 0,C 180,E1 -10032.09,E2 -10032.09} C_VEL
LIN {X 0,Y 574.974,Z 487.355,A -85,B 0,C 180,E1 -10035.575,E2 -10035.575} C_VEL
LIN {X 0,Y 576.754,Z 424.351,A -85,B 0,C 180,E1 -10036.486,E2 -10036.486} C_VEL
LIN {X 0,Y 566.099,Z 406.895,A -85,B 0,C 180,E1 -10037.909,E2 -10037.909} C_VEL
LIN {X 0,Y 553.282,Z 387.489,A -85,B 0,C 180,E1 -10039.72,E2 -10039.72} C_VEL
LIN {X 0,Y 544.456,Z 375.833,A -85,B 0,C 180,E1 -10041.023,E2 -10041.023} C_VEL
LIN {X 0,Y 541.053,Z 371.344,A -85,B 0,C 180,E1 -10041.547,E2 -10041.547} C_VEL
LIN {X 0,Y 537.278,Z 366.328,A -85,B 0,C 180,E1 -10042.144,E2 -10042.144} C_VEL
LIN {X 0,Y 534.433,Z 362.708,A -85,B 0,C 180,E1 -10042.601,E2 -10042.601} C_VEL
LIN {X 0,Y 533.576,Z 361.171,A -85,B 0,C 180,E1 -10042.75,E2 -10042.75} C_VEL
LIN {X 0,Y 530.914,Z 358.644,A -85,B 0,C 180,E1 -10043.171,E2 -10043.171} C_VEL
LIN {X 0,Y 529.721,Z 355.604,A -85,B 0,C 180,E1 -10043.404,E2 -10043.404} C_VEL
LIN {X 0,Y 529.662,Z 355.203,A -85,B 0,C 180,E1 -10043.422,E2 -10043.422} C_VEL
LIN {X 0,Y 529.628,Z 355.258,A -85,B 0,C 180,E1 -10046.756,E2 -10046.756} C_VEL
LIN {X 0,Y 529.669,Z 355.254,A -85,B 0,C 180,E1 -10050.108,E2 -10050.108} C_VEL
LIN {X 0,Y 529.646,Z 355.258,A -85,B 0,C 180,E1 -10053.301,E2 -10053.301} C_VEL
LIN {X 0,Y 529.631,Z 355.257,A -85,B 0,C 180,E1 -10056.761,E2 -10056.761} C_VEL
LIN {X 0,Y 529.686,Z 355.254,A -85,B 0,C 180,E1 -10060.064,E2 -10060.064} C_VEL
LIN {X 0,Y 529.634,Z 355.25,A -85,B 0,C 180,E1 -10063.324,E2 -10063.324} C_VEL
LIN {X 0,Y 529.631,Z 355.245,A -85,B 0,C 180,E1 -10066.795,E2 -10066.795} C_VEL
LIN {X 0,Y 529.681,Z 355.233,A -85,B 0,C 180,E1 -10070.108,E2 -10070.108} C_VEL
LIN {X 0,Y 529.627,Z 355.248,A -85,B 0,C 180,E1 -10073.387,E2 -10073.387} C_VEL
LIN {X 0,Y 529.638,Z 355.254,A -85,B 0,C 180,E1 -10076.862,E2 -10076.862} C_VEL
LIN {X 0,Y 529.69,Z 355.247,A -85,B 0,C 180,E1 -10080.216,E2 -10080.216} C_VEL
LIN {X 0,Y 529.627,Z 355.241,A -85,B 0,C 180,E1 -10083.572,E2 -10083.572} C_VEL
LIN {X 0,Y 529.634,Z 355.234,A -85,B 0,C 180,E1 -10087.049,E2 -10087.049} C_VEL
LIN {X 0,Y 529.667,Z 355.242,A -85,B 0,C 180,E1 -10090.221,E2 -10090.221} C_VEL
LIN {X 0,Y 529.625,Z 355.256,A -85,B 0,C 180,E1 -10093.539,E2 -10093.539} C_VEL
LIN {X 0,Y 529.669,Z 355.247,A -85,B 0,C 180,E1 -10096.844,E2 -10096.844} C_VEL
LIN {X 0,Y 529.64,Z 355.236,A -85,B 0,C 180,E1 -10100.096,E2 -10100.096} C_VEL
LIN {X 0,Y 529.627,Z 355.236,A -85,B 0,C 180,E1 -10103.475,E2 -10103.475} C_VEL
LIN {X 0,Y 529.683,Z 355.233,A -85,B 0,C 180,E1 -10106.762,E2 -10106.762} C_VEL
LIN {X 0,Y 529.629,Z 355.255,A -85,B 0,C 180,E1 -10110.02,E2 -10110.02} C_VEL
LIN {X 0,Y 529.64,Z 355.256,A -85,B 0,C 180,E1 -10113.454,E2 -10113.454} C_VEL
LIN {X 0,Y 529.685,Z 355.455,A -85,B 0,C 180,E1 -10116.576,E2 -10116.576} C_VEL
LIN {X 0,Y 531.295,Z 359.193,A -85,B 0,C 180,E1 -10117.301,E2 -10117.301} C_VEL
LIN {X 0,Y 536.976,Z 371.547,A -85,B 0,C 180,E1 -10119.591,E2 -10119.591} C_VEL
LIN {X 0,Y 550.839,Z 391.729,A -85,B 0,C 180,E1 -10121.739,E2 -10121.739} C_VEL
LIN {X 0,Y 562.562,Z 409.865,A -85,B 0,C 180,E1 -10123.425,E2 -10123.425} C_VEL
LIN {X 0,Y 574.643,Z 430.214,A -85,B 0,C 180,E1 -10125.069,E2 -10125.069} C_VEL
LIN {X 0,Y 576.866,Z 434.607,A -85,B 0,C 180,E1 -10125.369,E2 -10125.369} C_VEL
LIN {X 0,Y 569.179,Z 691.344,A -85,B 0,C 180,E1 -10128.984,E2 -10128.984} C_VEL
LIN {X 0,Y 566.9,Z 765.505,A -85,B 0,C 180,E1 -10130.043,E2 -10130.043} C_VEL
LIN {X 0,Y 565.176,Z 790.973,A -85,B 0,C 180,E1 -10130.566,E2 -10130.566} C_VEL
LIN {X 0,Y 563.236,Z 813.045,A -85,B 0,C 180,E1 -10131.177,E2 -10131.177} C_VEL
LIN {X 0,Y 560.692,Z 837.061,A -85,B 0,C 180,E1 -10132.03,E2 -10132.03} C_VEL
LIN {X 0,Y 558.175,Z 857.631,A -85,B 0,C 180,E1 -10132.93,E2 -10132.93} C_VEL
LIN {X 0,Y 555.075,Z 880.433,A -85,B 0,C 180,E1 -10134.115,E2 -10134.115} C_VEL
LIN {X 0,Y 552.1,Z 900.242,A -85,B 0,C 180,E1 -10135.342,E2 -10135.342} C_VEL
LIN {X 0,Y 549.066,Z 919.466,A -85,B 0,C 180,E1 -10136.707,E2 -10136.707} C_VEL
LIN {X 0,Y 545.654,Z 939.851,A -85,B 0,C 180,E1 -10138.393,E2 -10138.393} C_VEL
LIN {X 0,Y 542.725,Z 957.285,A -85,B 0,C 180,E1 -10140.048,E2 -10140.048} C_VEL
LIN {X 0,Y 539.48,Z 976.543,A -85,B 0,C 180,E1 -10142.156,E2 -10142.156} C_VEL
LIN {X 0,Y 536.998,Z 991.652,A -85,B 0,C 180,E1 -10144.051,E2 -10144.051} C_VEL
LIN {X 0,Y 534.392,Z 1008.386,A -85,B 0,C 180,E1 -10146.468,E2 -10146.468} C_VEL
LIN {X 0,Y 532.603,Z 1020.77,A -85,B 0,C 180,E1 -10148.526,E2 -10148.526} C_VEL
LIN {X 0,Y 530.883,Z 1034.172,A -85,B 0,C 180,E1 -10151.098,E2 -10151.098} C_VEL
LIN {X 0,Y 529.799,Z 1044.095,A -85,B 0,C 180,E1 -10153.329,E2 -10153.329} C_VEL
LIN {X 0,Y 528.928,Z 1053.815,A -85,B 0,C 180,E1 -10155.885,E2 -10155.885} C_VEL
LIN {X 0,Y 528.401,Z 1061.322,A -85,B 0,C 180,E1 -10158.318,E2 -10158.318} C_VEL
LIN {X 0,Y 528.114,Z 1067.163,A -85,B 0,C 180,E1 -10160.629,E2 -10160.629} C_VEL
LIN {X 0,Y 527.952,Z 1072.334,A -85,B 0,C 180,E1 -10163.366,E2 -10163.366} C_VEL
LIN {X 0,Y 527.922,Z 1075.175,A -85,B 0,C 180,E1 -10165.546,E2 -10165.546} C_VEL
LIN {X 0,Y 527.916,Z 1077.058,A -85,B 0,C 180,E1 -10167.938,E2 -10167.938} C_VEL
LIN {X 0,Y 527.908,Z 1077.492,A -85,B 0,C 180,E1 -10170.543,E2 -10170.543} C_VEL
LIN {X 0,Y 527.918,Z 1076.576,A -85,B 0,C 180,E1 -10172.823,E2 -10172.823} C_VEL
LIN {X 0,Y 527.935,Z 1074.252,A -85,B 0,C 180,E1 -10175.325,E2 -10175.325} C_VEL
LIN {X 0,Y 527.999,Z 1070.282,A -85,B 0,C 180,E1 -10177.837,E2 -10177.837} C_VEL
LIN {X 0,Y 528.179,Z 1065.365,A -85,B 0,C 180,E1 -10180.14,E2 -10180.14} C_VEL
LIN {X 0,Y 528.6,Z 1058.139,A -85,B 0,C 180,E1 -10182.786,E2 -10182.786} C_VEL
LIN {X 0,Y 529.215,Z 1050.208,A -85,B 0,C 180,E1 -10185.114,E2 -10185.114} C_VEL
LIN {X 0,Y 530.137,Z 1040.857,A -85,B 0,C 180,E1 -10187.451,E2 -10187.451} C_VEL
LIN {X 0,Y 531.499,Z 1029.162,A -85,B 0,C 180,E1 -10189.908,E2 -10189.908} C_VEL
LIN {X 0,Y 533.043,Z 1017.489,A -85,B 0,C 180,E1 -10192.034,E2 -10192.034} C_VEL
LIN {X 0,Y 535.335,Z 1001.832,A -85,B 0,C 180,E1 -10194.497,E2 -10194.497} C_VEL
LIN {X 0,Y 537.504,Z 987.941,A -85,B 0,C 180,E1 -10196.398,E2 -10196.398} C_VEL
LIN {X 0,Y 540.38,Z 970.296,A -85,B 0,C 180,E1 -10198.515,E2 -10198.515} C_VEL
LIN {X 0,Y 543.078,Z 953.791,A -85,B 0,C 180,E1 -10200.235,E2 -10200.235} C_VEL
LIN {X 0,Y 546.277,Z 934.581,A -85,B 0,C 180,E1 -10201.998,E2 -10201.998} C_VEL
LIN {X 0,Y 549.333,Z 915.171,A -85,B 0,C 180,E1 -10203.524,E2 -10203.524} C_VEL
LIN {X 0,Y 552.374,Z 895.308,A -85,B 0,C 180,E1 -10204.891,E2 -10204.891} C_VEL
LIN {X 0,Y 555.465,Z 873.063,A -85,B 0,C 180,E1 -10206.188,E2 -10206.188} C_VEL
LIN {X 0,Y 558.076,Z 853.029,A -85,B 0,C 180,E1 -10207.178,E2 -10207.178} C_VEL
LIN {X 0,Y 560.861,Z 828.542,A -85,B 0,C 180,E1 -10208.18,E2 -10208.18} C_VEL
LIN {X 0,Y 562.891,Z 807.673,A -85,B 0,C 180,E1 -10208.865,E2 -10208.865} C_VEL
LIN {X 0,Y 564.894,Z 783.094,A -85,B 0,C 180,E1 -10209.496,E2 -10209.496} C_VEL
LIN {X 0,Y 566.148,Z 759.815,A -85,B 0,C 180,E1 -10209.924,E2 -10209.924} C_VEL
LIN {X 0,Y 572.717,Z 523.949,A -85,B 0,C 180,E1 -10213.219,E2 -10213.219} C_VEL
LIN {X 0,Y 575.229,Z 433.455,A -85,B 0,C 180,E1 -10214.5,E2 -10214.5} C_VEL
LIN {X 0,Y 561.74,Z 410.227,A -85,B 0,C 180,E1 -10216.231,E2 -10216.231} C_VEL
LIN {X 0,Y 550.04,Z 391.577,A -85,B 0,C 180,E1 -10217.819,E2 -10217.819} C_VEL
LIN {X 0,Y 539.44,Z 375.609,A -85,B 0,C 180,E1 -10219.343,E2 -10219.343} C_VEL
LIN {X 0,Y 536.613,Z 371.19,A -85,B 0,C 180,E1 -10219.793,E2 -10219.793} C_VEL
LIN {X 0,Y 531.318,Z 359.259,A -85,B 0,C 180,E1 -10221.883,E2 -10221.883} C_VEL
LIN {X 0,Y 529.841,Z 356.307,A -85,B 0,C 180,E1 -10222.443,E2 -10222.443} C_VEL
LIN {X 0,Y 529.65,Z 355.241,A -85,B 0,C 180,E1 -10222.634,E2 -10222.634} C_VEL
LIN {X 0,Y 529.625,Z 355.242,A -85,B 0,C 180,E1 -10226.025,E2 -10226.025} C_VEL
LIN {X 0,Y 529.678,Z 355.232,A -85,B 0,C 180,E1 -10229.357,E2 -10229.357} C_VEL
LIN {X 0,Y 529.632,Z 355.234,A -85,B 0,C 180,E1 -10232.571,E2 -10232.571} C_VEL
LIN {X 0,Y 529.627,Z 355.237,A -85,B 0,C 180,E1 -10236.052,E2 -10236.052} C_VEL
LIN {X 0,Y 529.688,Z 355.248,A -85,B 0,C 180,E1 -10239.329,E2 -10239.329} C_VEL
LIN {X 0,Y 529.63,Z 355.253,A -85,B 0,C 180,E1 -10242.645,E2 -10242.645} C_VEL
LIN {X 0,Y 529.632,Z 355.235,A -85,B 0,C 180,E1 -10246.127,E2 -10246.127} C_VEL
LIN {X 0,Y 529.679,Z 355.235,A -85,B 0,C 180,E1 -10249.449,E2 -10249.449} C_VEL
LIN {X 0,Y 529.628,Z 355.256,A -85,B 0,C 180,E1 -10252.733,E2 -10252.733} C_VEL
LIN {X 0,Y 529.646,Z 355.231,A -85,B 0,C 180,E1 -10256.103,E2 -10256.103} C_VEL
LIN {X 0,Y 529.662,Z 355.244,A -85,B 0,C 180,E1 -10259.351,E2 -10259.351} C_VEL
LIN {X 0,Y 529.627,Z 355.256,A -85,B 0,C 180,E1 -10262.705,E2 -10262.705} C_VEL
LIN {X 0,Y 529.667,Z 355.226,A -85,B 0,C 180,E1 -10266.068,E2 -10266.068} C_VEL
LIN {X 0,Y 529.638,Z 355.254,A -85,B 0,C 180,E1 -10269.234,E2 -10269.234} C_VEL
LIN {X 0,Y 529.632,Z 355.248,A -85,B 0,C 180,E1 -10272.65,E2 -10272.65} C_VEL
LIN {X 0,Y 529.685,Z 355.227,A -85,B 0,C 180,E1 -10275.886,E2 -10275.886} C_VEL
LIN {X 0,Y 529.631,Z 355.254,A -85,B 0,C 180,E1 -10279.178,E2 -10279.178} C_VEL
LIN {X 0,Y 529.645,Z 355.254,A -85,B 0,C 180,E1 -10282.651,E2 -10282.651} C_VEL
LIN {X 0,Y 529.677,Z 355.229,A -85,B 0,C 180,E1 -10285.974,E2 -10285.974} C_VEL
LIN {X 0,Y 529.628,Z 355.235,A -85,B 0,C 180,E1 -10289.273,E2 -10289.273} C_VEL
LIN {X 0,Y 529.657,Z 355.238,A -85,B 0,C 180,E1 -10292.652,E2 -10292.652} C_VEL
LIN {X 0,Y 529.663,Z 355.244,A -85,B 0,C 180,E1 -10295.952,E2 -10295.952} C_VEL
LIN {X 0,Y 529.629,Z 355.248,A -85,B 0,C 180,E1 -10299.282,E2 -10299.282} C_VEL
LIN {X 0,Y 529.658,Z 355.461,A -85,B 0,C 180,E1 -10301.46,E2 -10301.46} C_VEL
LIN {X 0,Y 530.843,Z 358.59,A -85,B 0,C 180,E1 -10301.676,E2 -10301.676} C_VEL
LIN {X 0,Y 533.807,Z 361.718,A -85,B 0,C 180,E1 -10302.112,E2 -10302.112} C_VEL
LIN {X 0,Y 536.407,Z 365.576,A -85,B 0,C 180,E1 -10302.51,E2 -10302.51} C_VEL
LIN {X 0,Y 538.037,Z 367.623,A -85,B 0,C 180,E1 -10302.749,E2 -10302.749} C_VEL
LIN {X 0,Y 545.712,Z 378.039,A -85,B 0,C 180,E1 -10303.855,E2 -10303.855} C_VEL
LIN {X 0,Y 556.144,Z 392.807,A -85,B 0,C 180,E1 -10305.286,E2 -10305.286} C_VEL
LIN {X 0,Y 570.491,Z 415.87,A -85,B 0,C 180,E1 -10307.162,E2 -10307.162} C_VEL
LIN {X 0,Y 575.39,Z 424.466,A -85,B 0,C 180,E1 -10307.781,E2 -10307.781} C_VEL
LIN {X 0,Y 568.361,Z 671.373,A -85,B 0,C 180,E1 -10311.233,E2 -10311.233} C_VEL
LIN {X 0,Y 566.25,Z 742.43,A -85,B 0,C 180,E1 -10312.242,E2 -10312.242} C_VEL
LIN {X 0,Y 565.216,Z 760.968,A -85,B 0,C 180,E1 -10312.606,E2 -10312.606} C_VEL
LIN {X 0,Y 563.976,Z 768.571,A -85,B 0,C 180,E1 -10312.713,E2 -10312.713} C_VEL
LIN {X 0,Y 557.724,Z 787.631,A -85,B 0,C 180,E1 -10312.862,E2 -10312.862} C_VEL
LIN {X 0,Y 556.189,Z 795.001,A -85,B 0,C 180,E1 -10313.048,E2 -10313.048} C_VEL
LIN {X 0,Y 553.823,Z 816.925,A -85,B 0,C 180,E1 -10313.88,E2 -10313.88} C_VEL
LIN {X 0,Y 551.238,Z 837.98,A -85,B 0,C 180,E1 -10314.836,E2 -10314.836} C_VEL
LIN {X 0,Y 548.084,Z 860.394,A -85,B 0,C 180,E1 -10316.065,E2 -10316.065} C_VEL
LIN {X 0,Y 545.126,Z 879.682,A -85,B 0,C 180,E1 -10317.304,E2 -10317.304} C_VEL
LIN {X 0,Y 541.516,Z 901.62,A -85,B 0,C 180,E1 -10318.955,E2 -10318.955} C_VEL
LIN {X 0,Y 538.535,Z 918.916,A -85,B 0,C 180,E1 -10320.464,E2 -10320.464} C_VEL
LIN {X 0,Y 535.012,Z 938.668,A -85,B 0,C 180,E1 -10322.448,E2 -10322.448} C_VEL
LIN {X 0,Y 532.343,Z 953.518,A -85,B 0,C 180,E1 -10324.166,E2 -10324.166} C_VEL
LIN {X 0,Y 529.529,Z 969.671,A -85,B 0,C 180,E1 -10326.284,E2 -10326.284} C_VEL
LIN {X 0,Y 527.011,Z 984.287,A -85,B 0,C 180,E1 -10328.52,E2 -10328.52} C_VEL
LIN {X 0,Y 524.903,Z 997.776,A -85,B 0,C 180,E1 -10330.881,E2 -10330.881} C_VEL
LIN {X 0,Y 523.254,Z 1009.144,A -85,B 0,C 180,E1 -10333.229,E2 -10333.229} C_VEL
LIN {X 0,Y 522.018,Z 1019.015,A -85,B 0,C 180,E1 -10335.581,E2 -10335.581} C_VEL
LIN {X 0,Y 521.073,Z 1027.98,A -85,B 0,C 180,E1 -10338.152,E2 -10338.152} C_VEL
LIN {X 0,Y 520.512,Z 1034.725,A -85,B 0,C 180,E1 -10340.491,E2 -10340.491} C_VEL
LIN {X 0,Y 520.15,Z 1040.86,A -85,B 0,C 180,E1 -10343.155,E2 -10343.155} C_VEL
LIN {X 0,Y 519.998,Z 1044.948,A -85,B 0,C 180,E1 -10345.589,E2 -10345.589} C_VEL
LIN {X 0,Y 519.945,Z 1047.789,A -85,B 0,C 180,E1 -10348.016,E2 -10348.016} C_VEL
LIN {X 0,Y 519.924,Z 1049.378,A -85,B 0,C 180,E1 -10350.771,E2 -10350.771} C_VEL
LIN {X 0,Y 519.92,Z 1049.427,A -85,B 0,C 180,E1 -10353.087,E2 -10353.087} C_VEL
LIN {X 0,Y 519.94,Z 1048.133,A -85,B 0,C 180,E1 -10355.739,E2 -10355.739} C_VEL
LIN {X 0,Y 519.999,Z 1045.254,A -85,B 0,C 180,E1 -10358.292,E2 -10358.292} C_VEL
LIN {X 0,Y 520.127,Z 1041.42,A -85,B 0,C 180,E1 -10360.635,E2 -10360.635} C_VEL
LIN {X 0,Y 520.489,Z 1035.167,A -85,B 0,C 180,E1 -10363.441,E2 -10363.441} C_VEL
LIN {X 0,Y 521.042,Z 1028.406,A -85,B 0,C 180,E1 -10365.813,E2 -10365.813} C_VEL
LIN {X 0,Y 521.993,Z 1019.423,A -85,B 0,C 180,E1 -10368.425,E2 -10368.425} C_VEL
LIN {X 0,Y 523.276,Z 1009.231,A -85,B 0,C 180,E1 -10370.868,E2 -10370.868} C_VEL
LIN {X 0,Y 525.083,Z 997.044,A -85,B 0,C 180,E1 -10373.386,E2 -10373.386} C_VEL
LIN {X 0,Y 527.237,Z 983.565,A -85,B 0,C 180,E1 -10375.74,E2 -10375.74} C_VEL
LIN {X 0,Y 529.889,Z 968.582,A -85,B 0,C 180,E1 -10378.025,E2 -10378.025} C_VEL
LIN {X 0,Y 532.701,Z 952.868,A -85,B 0,C 180,E1 -10380.082,E2 -10380.082} C_VEL
LIN {X 0,Y 535.922,Z 935.701,A -85,B 0,C 180,E1 -10382.06,E2 -10382.06} C_VEL
LIN {X 0,Y 539.214,Z 917.432,A -85,B 0,C 180,E1 -10383.865,E2 -10383.865} C_VEL
LIN {X 0,Y 542.562,Z 898.714,A -85,B 0,C 180,E1 -10385.487,E2 -10385.487} C_VEL
LIN {X 0,Y 546.058,Z 877.896,A -85,B 0,C 180,E1 -10387.026,E2 -10387.026} C_VEL
LIN {X 0,Y 549.092,Z 858.675,A -85,B 0,C 180,E1 -10388.253,E2 -10388.253} C_VEL
LIN {X 0,Y 552.425,Z 835.335,A -85,B 0,C 180,E1 -10389.51,E2 -10389.51} C_VEL
LIN {X 0,Y 554.858,Z 816.079,A -85,B 0,C 180,E1 -10390.379,E2 -10390.379} C_VEL
LIN {X 0,Y 557.403,Z 793.074,A -85,B 0,C 180,E1 -10391.244,E2 -10391.244} C_VEL
LIN {X 0,Y 559.415,Z 769.948,A -85,B 0,C 180,E1 -10391.916,E2 -10391.916} C_VEL
LIN {X 0,Y 560.948,Z 747.908,A -85,B 0,C 180,E1 -10392.407,E2 -10392.407} C_VEL
LIN {X 0,Y 562.272,Z 713.265,A -85,B 0,C 180,E1 -10392.942,E2 -10392.942} C_VEL
LIN {X 0,Y 570.155,Z 460.552,A -85,B 0,C 180,E1 -10396.523,E2 -10396.523} C_VEL
LIN {X 0,Y 571.092,Z 427.886,A -85,B 0,C 180,E1 -10397.003,E2 -10397.003} C_VEL
LIN {X 0,Y 561.305,Z 411.868,A -85,B 0,C 180,E1 -10398.342,E2 -10398.342} C_VEL
LIN {X 0,Y 549.264,Z 393.528,A -85,B 0,C 180,E1 -10400.081,E2 -10400.081} C_VEL
LIN {X 0,Y 537.715,Z 378.063,A -85,B 0,C 180,E1 -10401.842,E2 -10401.842} C_VEL
LIN {X 0,Y 533.399,Z 372.513,A -85,B 0,C 180,E1 -10402.533,E2 -10402.533} C_VEL
LIN {X 0,Y 529.57,Z 367.488,A -85,B 0,C 180,E1 -10403.167,E2 -10403.167} C_VEL
LIN {X 0,Y 526.719,Z 363.943,A -85,B 0,C 180,E1 -10403.647,E2 -10403.647} C_VEL
LIN {X 0,Y 525.546,Z 362.05,A -85,B 0,C 180,E1 -10403.857,E2 -10403.857} C_VEL
LIN {X 0,Y 522.876,Z 359.479,A -85,B 0,C 180,E1 -10404.304,E2 -10404.304} C_VEL
LIN {X 0,Y 521.712,Z 356.383,A -85,B 0,C 180,E1 -10404.546,E2 -10404.546} C_VEL
LIN {X 0,Y 521.747,Z 356.229,A -85,B 0,C 180,E1 -10407.807,E2 -10407.807} C_VEL
LIN {X 0,Y 521.692,Z 356.236,A -85,B 0,C 180,E1 -10410.993,E2 -10410.993} C_VEL
LIN {X 0,Y 521.703,Z 356.229,A -85,B 0,C 180,E1 -10414.454,E2 -10414.454} C_VEL
LIN {X 0,Y 521.748,Z 356.225,A -85,B 0,C 180,E1 -10417.819,E2 -10417.819} C_VEL
LIN {X 0,Y 521.69,Z 356.239,A -85,B 0,C 180,E1 -10421.1,E2 -10421.1} C_VEL
LIN {X 0,Y 521.704,Z 356.242,A -85,B 0,C 180,E1 -10424.588,E2 -10424.588} C_VEL
LIN {X 0,Y 521.728,Z 356.242,A -85,B 0,C 180,E1 -10427.83,E2 -10427.83} C_VEL
LIN {X 0,Y 521.686,Z 356.238,A -85,B 0,C 180,E1 -10431.18,E2 -10431.18} C_VEL
LIN {X 0,Y 521.724,Z 356.222,A -85,B 0,C 180,E1 -10434.501,E2 -10434.501} C_VEL
LIN {X 0,Y 521.708,Z 356.23,A -85,B 0,C 180,E1 -10437.803,E2 -10437.803} C_VEL
LIN {X 0,Y 521.689,Z 356.245,A -85,B 0,C 180,E1 -10441.208,E2 -10441.208} C_VEL
LIN {X 0,Y 521.734,Z 356.243,A -85,B 0,C 180,E1 -10444.617,E2 -10444.617} C_VEL
LIN {X 0,Y 521.704,Z 356.226,A -85,B 0,C 180,E1 -10447.932,E2 -10447.932} C_VEL
LIN {X 0,Y 521.685,Z 356.223,A -85,B 0,C 180,E1 -10451.386,E2 -10451.386} C_VEL
LIN {X 0,Y 521.735,Z 356.222,A -85,B 0,C 180,E1 -10454.767,E2 -10454.767} C_VEL
LIN {X 0,Y 521.705,Z 356.239,A -85,B 0,C 180,E1 -10458.089,E2 -10458.089} C_VEL
LIN {X 0,Y 521.689,Z 356.245,A -85,B 0,C 180,E1 -10461.474,E2 -10461.474} C_VEL
LIN {X 0,Y 521.746,Z 356.234,A -85,B 0,C 180,E1 -10464.717,E2 -10464.717} C_VEL
LIN {X 0,Y 521.691,Z 356.236,A -85,B 0,C 180,E1 -10468.007,E2 -10468.007} C_VEL
LIN {X 0,Y 521.693,Z 356.244,A -85,B 0,C 180,E1 -10471.55,E2 -10471.55} C_VEL
LIN {X 0,Y 521.744,Z 356.239,A -85,B 0,C 180,E1 -10474.892,E2 -10474.892} C_VEL
LIN {X 0,Y 521.704,Z 356.277,A -85,B 0,C 180,E1 -10475.502,E2 -10475.502} C_VEL
LIN {X 0,Y 522.774,Z 359.385,A -85,B 0,C 180,E1 -10476.093,E2 -10476.093} C_VEL
LIN {X 0,Y 523.933,Z 361.432,A -85,B 0,C 180,E1 -10476.544,E2 -10476.544} C_VEL
LIN {X 0,Y 528.434,Z 371.168,A -85,B 0,C 180,E1 -10478.42,E2 -10478.42} C_VEL
LIN {X 0,Y 539.128,Z 386.343,A -85,B 0,C 180,E1 -10480.178,E2 -10480.178} C_VEL
LIN {X 0,Y 550.523,Z 403.277,A -85,B 0,C 180,E1 -10481.925,E2 -10481.925} C_VEL
LIN {X 0,Y 563.726,Z 424.56,A -85,B 0,C 180,E1 -10483.822,E2 -10483.822} C_VEL
LIN {X 0,Y 571.142,Z 437.721,A -85,B 0,C 180,E1 -10484.842,E2 -10484.842} C_VEL
LIN {X 0,Y 563.156,Z 693.159,A -85,B 0,C 180,E1 -10488.468,E2 -10488.468} C_VEL
LIN {X 0,Y 560.832,Z 765.394,A -85,B 0,C 180,E1 -10489.509,E2 -10489.509} C_VEL
LIN {X 0,Y 559.048,Z 790.818,A -85,B 0,C 180,E1 -10490.035,E2 -10490.035} C_VEL
LIN {X 0,Y 557.042,Z 812.768,A -85,B 0,C 180,E1 -10490.646,E2 -10490.646} C_VEL
LIN {X 0,Y 554.339,Z 837.207,A -85,B 0,C 180,E1 -10491.521,E2 -10491.521} C_VEL
LIN {X 0,Y 551.734,Z 857.654,A -85,B 0,C 180,E1 -10492.423,E2 -10492.423} C_VEL
LIN {X 0,Y 548.527,Z 880.226,A -85,B 0,C 180,E1 -10493.605,E2 -10493.605} C_VEL
LIN {X 0,Y 545.4,Z 900.192,A -85,B 0,C 180,E1 -10494.854,E2 -10494.854} C_VEL
LIN {X 0,Y 542.016,Z 920.757,A -85,B 0,C 180,E1 -10496.334,E2 -10496.334} C_VEL
LIN {X 0,Y 538.552,Z 940.361,A -85,B 0,C 180,E1 -10497.99,E2 -10497.99} C_VEL
LIN {X 0,Y 535.489,Z 957.728,A -85,B 0,C 180,E1 -10499.663,E2 -10499.663} C_VEL
LIN {X 0,Y 532.179,Z 976.406,A -85,B 0,C 180,E1 -10501.74,E2 -10501.74} C_VEL
LIN {X 0,Y 529.558,Z 991.503,A -85,B 0,C 180,E1 -10503.659,E2 -10503.659} C_VEL
LIN {X 0,Y 526.877,Z 1007.787,A -85,B 0,C 180,E1 -10506.039,E2 -10506.039} C_VEL
LIN {X 0,Y 524.906,Z 1020.594,A -85,B 0,C 180,E1 -10508.195,E2 -10508.195} C_VEL
LIN {X 0,Y 523.082,Z 1033.981,A -85,B 0,C 180,E1 -10510.805,E2 -10510.805} C_VEL
LIN {X 0,Y 521.928,Z 1043.894,A -85,B 0,C 180,E1 -10513.07,E2 -10513.07} C_VEL
LIN {X 0,Y 520.997,Z 1053.602,A -85,B 0,C 180,E1 -10515.666,E2 -10515.666} C_VEL
LIN {X 0,Y 520.436,Z 1061.105,A -85,B 0,C 180,E1 -10518.137,E2 -10518.137} C_VEL
LIN {X 0,Y 520.118,Z 1067.204,A -85,B 0,C 180,E1 -10520.595,E2 -10520.595} C_VEL
LIN {X 0,Y 519.957,Z 1072.119,A -85,B 0,C 180,E1 -10523.263,E2 -10523.263} C_VEL
LIN {X 0,Y 519.925,Z 1074.96,A -85,B 0,C 180,E1 -10525.478,E2 -10525.478} C_VEL
LIN {X 0,Y 519.918,Z 1076.844,A -85,B 0,C 180,E1 -10527.906,E2 -10527.906} C_VEL
LIN {X 0,Y 519.911,Z 1077.278,A -85,B 0,C 180,E1 -10530.551,E2 -10530.551} C_VEL
LIN {X 0,Y 519.922,Z 1076.363,A -85,B 0,C 180,E1 -10532.866,E2 -10532.866} C_VEL
LIN {X 0,Y 519.938,Z 1074.038,A -85,B 0,C 180,E1 -10535.407,E2 -10535.407} C_VEL
LIN {X 0,Y 520.01,Z 1069.984,A -85,B 0,C 180,E1 -10538.002,E2 -10538.002} C_VEL
LIN {X 0,Y 520.199,Z 1065.15,A -85,B 0,C 180,E1 -10540.297,E2 -10540.297} C_VEL
LIN {X 0,Y 520.65,Z 1057.92,A -85,B 0,C 180,E1 -10542.985,E2 -10542.985} C_VEL
LIN {X 0,Y 521.303,Z 1049.98,A -85,B 0,C 180,E1 -10545.349,E2 -10545.349} C_VEL
LIN {X 0,Y 522.339,Z 1040.151,A -85,B 0,C 180,E1 -10547.835,E2 -10547.835} C_VEL
LIN {X 0,Y 523.794,Z 1028.323,A -85,B 0,C 180,E1 -10550.33,E2 -10550.33} C_VEL
LIN {X 0,Y 525.579,Z 1015.933,A -85,B 0,C 180,E1 -10552.6,E2 -10552.6} C_VEL
LIN {X 0,Y 527.911,Z 1000.767,A -85,B 0,C 180,E1 -10554.984,E2 -10554.984} C_VEL
LIN {X 0,Y 530.228,Z 986.789,A -85,B 0,C 180,E1 -10556.91,E2 -10556.91} C_VEL
LIN {X 0,Y 533.358,Z 968.372,A -85,B 0,C 180,E1 -10559.118,E2 -10559.118} C_VEL
LIN {X 0,Y 536.241,Z 951.777,A -85,B 0,C 180,E1 -10560.849,E2 -10560.849} C_VEL
LIN {X 0,Y 539.87,Z 930.52,A -85,B 0,C 180,E1 -10562.769,E2 -10562.769} C_VEL
LIN {X 0,Y 542.847,Z 912.461,A -85,B 0,C 180,E1 -10564.18,E2 -10564.18} C_VEL
LIN {X 0,Y 546.432,Z 889.637,A -85,B 0,C 180,E1 -10565.713,E2 -10565.713} C_VEL
LIN {X 0,Y 549.283,Z 869.832,A -85,B 0,C 180,E1 -10566.84,E2 -10566.84} C_VEL
LIN {X 0,Y 552.341,Z 846.958,A -85,B 0,C 180,E1 -10567.943,E2 -10567.943} C_VEL
LIN {X 0,Y 554.746,Z 825.697,A -85,B 0,C 180,E1 -10568.781,E2 -10568.781} C_VEL
LIN {X 0,Y 556.812,Z 805.071,A -85,B 0,C 180,E1 -10569.448,E2 -10569.448} C_VEL
LIN {X 0,Y 558.849,Z 779.526,A -85,B 0,C 180,E1 -10570.081,E2 -10570.081} C_VEL
LIN {X 0,Y 560.029,Z 757.601,A -85,B 0,C 180,E1 -10570.474,E2 -10570.474} C_VEL
LIN {X 0,Y 567.099,Z 514.322,A -85,B 0,C 180,E1 -10573.899,E2 -10573.899} C_VEL
LIN {X 0,Y 569.298,Z 436.665,A -85,B 0,C 180,E1 -10575.014,E2 -10575.014} C_VEL
LIN {X 0,Y 555.161,Z 412.311,A -85,B 0,C 180,E1 -10576.881,E2 -10576.881} C_VEL
LIN {X 0,Y 543.462,Z 393.751,A -85,B 0,C 180,E1 -10578.521,E2 -10578.521} C_VEL
LIN {X 0,Y 531.779,Z 376.417,A -85,B 0,C 180,E1 -10580.261,E2 -10580.261} C_VEL
LIN {X 0,Y 527.94,Z 370.718,A -85,B 0,C 180,E1 -10580.899,E2 -10580.899} C_VEL
LIN {X 0,Y 524.841,Z 363.754,A -85,B 0,C 180,E1 -10582.16,E2 -10582.16} C_VEL
LIN {X 0,Y 522.901,Z 359.486,A -85,B 0,C 180,E1 -10582.962,E2 -10582.962} C_VEL
LIN {X 0,Y 521.706,Z 356.235,A -85,B 0,C 180,E1 -10583.549,E2 -10583.549} C_VEL
LIN {X 0,Y 521.731,Z 356.236,A -85,B 0,C 180,E1 -10586.893,E2 -10586.893} C_VEL
LIN {X 0,Y 521.686,Z 356.24,A -85,B 0,C 180,E1 -10590.255,E2 -10590.255} C_VEL
LIN {X 0,Y 521.719,Z 356.226,A -85,B 0,C 180,E1 -10593.6,E2 -10593.6} C_VEL
LIN {X 0,Y 521.715,Z 356.218,A -85,B 0,C 180,E1 -10596.917,E2 -10596.917} C_VEL
LIN {X 0,Y 521.685,Z 356.228,A -85,B 0,C 180,E1 -10600.286,E2 -10600.286} C_VEL
LIN {X 0,Y 521.733,Z 356.241,A -85,B 0,C 180,E1 -10603.637,E2 -10603.637} C_VEL
LIN {X 0,Y 521.695,Z 356.234,A -85,B 0,C 180,E1 -10606.816,E2 -10606.816} C_VEL
LIN {X 0,Y 521.689,Z 356.217,A -85,B 0,C 180,E1 -10610.29,E2 -10610.29} C_VEL
LIN {X 0,Y 521.752,Z 356.237,A -85,B 0,C 180,E1 -10613.618,E2 -10613.618} C_VEL
LIN {X 0,Y 521.699,Z 356.235,A -85,B 0,C 180,E1 -10617.034,E2 -10617.034} C_VEL
LIN {X 0,Y 521.69,Z 356.216,A -85,B 0,C 180,E1 -10620.439,E2 -10620.439} C_VEL
LIN {X 0,Y 521.743,Z 356.242,A -85,B 0,C 180,E1 -10623.736,E2 -10623.736} C_VEL
LIN {X 0,Y 521.691,Z 356.229,A -85,B 0,C 180,E1 -10627.046,E2 -10627.046} C_VEL
LIN {X 0,Y 521.696,Z 356.219,A -85,B 0,C 180,E1 -10630.51,E2 -10630.51} C_VEL
LIN {X 0,Y 521.751,Z 356.241,A -85,B 0,C 180,E1 -10633.86,E2 -10633.86} C_VEL
LIN {X 0,Y 521.691,Z 356.23,A -85,B 0,C 180,E1 -10637.167,E2 -10637.167} C_VEL
LIN {X 0,Y 521.7,Z 356.22,A -85,B 0,C 180,E1 -10640.65,E2 -10640.65} C_VEL
LIN {X 0,Y 521.738,Z 356.235,A -85,B 0,C 180,E1 -10643.915,E2 -10643.915} C_VEL
LIN {X 0,Y 521.694,Z 356.246,A -85,B 0,C 180,E1 -10647.263,E2 -10647.263} C_VEL
LIN {X 0,Y 521.715,Z 356.232,A -85,B 0,C 180,E1 -10650.651,E2 -10650.651} C_VEL
LIN {X 0,Y 521.734,Z 356.225,A -85,B 0,C 180,E1 -10654.029,E2 -10654.029} C_VEL
LIN {X 0,Y 521.691,Z 356.234,A -85,B 0,C 180,E1 -10657.414,E2 -10657.414} C_VEL
LIN {X 0,Y 521.778,Z 356.399,A -85,B 0,C 180,E1 -10660.442,E2 -10660.442} C_VEL
LIN {X 0,Y 522.979,Z 359.628,A -85,B 0,C 180,E1 -10660.672,E2 -10660.672} C_VEL
LIN {X 0,Y 525.944,Z 362.848,A -85,B 0,C 180,E1 -10661.132,E2 -10661.132} C_VEL
LIN {X 0,Y 528.492,Z 366.593,A -85,B 0,C 180,E1 -10661.54,E2 -10661.54} C_VEL
LIN {X 0,Y 530.32,Z 368.719,A -85,B 0,C 180,E1 -10661.816,E2 -10661.816} C_VEL
LIN {X 0,Y 541.639,Z 384.042,A -85,B 0,C 180,E1 -10663.498,E2 -10663.498} C_VEL
LIN {X 0,Y 551.99,Z 398.851,A -85,B 0,C 180,E1 -10664.948,E2 -10664.948} C_VEL
LIN {X 0,Y 565.842,Z 421.277,A -85,B 0,C 180,E1 -10666.797,E2 -10666.797} C_VEL
LIN {X 0,Y 569.505,Z 427.95,A -85,B 0,C 180,E1 -10667.274,E2 -10667.274} C_VEL
LIN {X 0,Y 562.193,Z 673.756,A -85,B 0,C 180,E1 -10670.739,E2 -10670.739} C_VEL
LIN {X 0,Y 560.05,Z 742.763,A -85,B 0,C 180,E1 -10671.729,E2 -10671.729} C_VEL
LIN {X 0,Y 558.494,Z 767.605,A -85,B 0,C 180,E1 -10672.253,E2 -10672.253} C_VEL
LIN {X 0,Y 556.702,Z 789.074,A -85,B 0,C 180,E1 -10672.857,E2 -10672.857} C_VEL
LIN {X 0,Y 556.189,Z 795.001,A -85,B 0,C 180,E1 -10673.048,E2 -10673.048} C_VEL
LIN {X 0,Y 554.625,Z 802.402,A -85,B 0,C 180,E1 -10673.249,E2 -10673.249} C_VEL
LIN {X 0,Y 547.803,Z 821.03,A -85,B 0,C 180,E1 -10673.591,E2 -10673.591} C_VEL
LIN {X 0,Y 546.087,Z 828.142,A -85,B 0,C 180,E1 -10673.849,E2 -10673.849} C_VEL
LIN {X 0,Y 543.236,Z 848.713,A -85,B 0,C 180,E1 -10674.887,E2 -10674.887} C_VEL
LIN {X 0,Y 539.955,Z 870.722,A -85,B 0,C 180,E1 -10676.198,E2 -10676.198} C_VEL
LIN {X 0,Y 536.621,Z 890.593,A -85,B 0,C 180,E1 -10677.602,E2 -10677.602} C_VEL
LIN {X 0,Y 533.176,Z 910.358,A -85,B 0,C 180,E1 -10679.205,E2 -10679.205} C_VEL
LIN {X 0,Y 529.69,Z 929.02,A -85,B 0,C 180,E1 -10680.979,E2 -10680.979} C_VEL
LIN {X 0,Y 526.501,Z 946.269,A -85,B 0,C 180,E1 -10682.85,E2 -10682.85} C_VEL
LIN {X 0,Y 523.41,Z 962.637,A -85,B 0,C 180,E1 -10684.907,E2 -10684.907} C_VEL
LIN {X 0,Y 520.952,Z 976.127,A -85,B 0,C 180,E1 -10686.835,E2 -10686.835} C_VEL
LIN {X 0,Y 518.32,Z 991.274,A -85,B 0,C 180,E1 -10689.328,E2 -10689.328} C_VEL
LIN {X 0,Y 516.488,Z 1002.577,A -85,B 0,C 180,E1 -10691.489,E2 -10691.489} C_VEL
LIN {X 0,Y 514.852,Z 1014.038,A -85,B 0,C 180,E1 -10694.016,E2 -10694.016} C_VEL
LIN {X 0,Y 513.683,Z 1023.402,A -85,B 0,C 180,E1 -10696.492,E2 -10696.492} C_VEL
LIN {X 0,Y 512.857,Z 1031.735,A -85,B 0,C 180,E1 -10699.099,E2 -10699.099} C_VEL
LIN {X 0,Y 512.332,Z 1038.256,A -85,B 0,C 180,E1 -10701.696,E2 -10701.696} C_VEL
LIN {X 0,Y 512.085,Z 1042.948,A -85,B 0,C 180,E1 -10704.06,E2 -10704.06} C_VEL
LIN {X 0,Y 511.961,Z 1046.921,A -85,B 0,C 180,E1 -10706.865,E2 -10706.865} C_VEL
LIN {X 0,Y 511.926,Z 1048.902,A -85,B 0,C 180,E1 -10709.217,E2 -10709.217} C_VEL
LIN {X 0,Y 511.909,Z 1049.755,A -85,B 0,C 180,E1 -10711.567,E2 -10711.567} C_VEL
LIN {X 0,Y 511.927,Z 1049.208,A -85,B 0,C 180,E1 -10714.369,E2 -10714.369} C_VEL
LIN {X 0,Y 511.958,Z 1047.422,A -85,B 0,C 180,E1 -10716.73,E2 -10716.73} C_VEL
LIN {X 0,Y 512.054,Z 1044.168,A -85,B 0,C 180,E1 -10719.327,E2 -10719.327} C_VEL
LIN {X 0,Y 512.293,Z 1039.036,A -85,B 0,C 180,E1 -10722.055,E2 -10722.055} C_VEL
LIN {X 0,Y 512.728,Z 1033.212,A -85,B 0,C 180,E1 -10724.455,E2 -10724.455} C_VEL
LIN {X 0,Y 513.59,Z 1024.442,A -85,B 0,C 180,E1 -10727.33,E2 -10727.33} C_VEL
LIN {X 0,Y 514.634,Z 1015.897,A -85,B 0,C 180,E1 -10729.641,E2 -10729.641} C_VEL
LIN {X 0,Y 516.32,Z 1004.278,A -85,B 0,C 180,E1 -10732.307,E2 -10732.307} C_VEL
LIN {X 0,Y 518.132,Z 992.986,A -85,B 0,C 180,E1 -10734.513,E2 -10734.513} C_VEL
LIN {X 0,Y 520.574,Z 979.45,A -85,B 0,C 180,E1 -10736.832,E2 -10736.832} C_VEL
LIN {X 0,Y 523.326,Z 964.419,A -85,B 0,C 180,E1 -10739.032,E2 -10739.032} C_VEL
LIN {X 0,Y 526.471,Z 948.321,A -85,B 0,C 180,E1 -10741.104,E2 -10741.104} C_VEL
LIN {X 0,Y 529.883,Z 930.385,A -85,B 0,C 180,E1 -10743.088,E2 -10743.088} C_VEL
LIN {X 0,Y 533.251,Z 912.846,A -85,B 0,C 180,E1 -10744.786,E2 -10744.786} C_VEL
LIN {X 0,Y 536.905,Z 892.908,A -85,B 0,C 180,E1 -10746.447,E2 -10746.447} C_VEL
LIN {X 0,Y 539.99,Z 875.14,A -85,B 0,C 180,E1 -10747.733,E2 -10747.733} C_VEL
LIN {X 0,Y 543.416,Z 853.979,A -85,B 0,C 180,E1 -10749.06,E2 -10749.06} C_VEL
LIN {X 0,Y 546.462,Z 832.874,A -85,B 0,C 180,E1 -10750.165,E2 -10750.165} C_VEL
LIN {X 0,Y 549.328,Z 810.672,A -85,B 0,C 180,E1 -10751.148,E2 -10751.148} C_VEL
LIN {X 0,Y 551.828,Z 786.94,A -85,B 0,C 180,E1 -10751.982,E2 -10751.982} C_VEL
LIN {X 0,Y 553.848,Z 764.046,A -85,B 0,C 180,E1 -10752.615,E2 -10752.615} C_VEL
LIN {X 0,Y 555.383,Z 739.151,A -85,B 0,C 180,E1 -10753.108,E2 -10753.108} C_VEL
LIN {X 0,Y 563.128,Z 502.46,A -85,B 0,C 180,E1 -10756.503,E2 -10756.503} C_VEL
LIN {X 0,Y 565.416,Z 431.39,A -85,B 0,C 180,E1 -10757.538,E2 -10757.538} C_VEL
LIN {X 0,Y 556.326,Z 416.472,A -85,B 0,C 180,E1 -10758.815,E2 -10758.815} C_VEL
LIN {X 0,Y 545.269,Z 399.555,A -85,B 0,C 180,E1 -10760.448,E2 -10760.448} C_VEL
LIN {X 0,Y 533.928,Z 384.264,A -85,B 0,C 180,E1 -10762.214,E2 -10762.214} C_VEL
LIN {X 0,Y 529.276,Z 378.296,A -85,B 0,C 180,E1 -10762.974,E2 -10762.974} C_VEL
LIN {X 0,Y 525.892,Z 373.843,A -85,B 0,C 180,E1 -10763.547,E2 -10763.547} C_VEL
LIN {X 0,Y 522.705,Z 369.46,A -85,B 0,C 180,E1 -10764.104,E2 -10764.104} C_VEL
LIN {X 0,Y 519.096,Z 365.359,A -85,B 0,C 180,E1 -10764.733,E2 -10764.733} C_VEL
LIN {X 0,Y 517.978,Z 363.279,A -85,B 0,C 180,E1 -10764.95,E2 -10764.95} C_VEL
LIN {X 0,Y 515.291,Z 360.955,A -85,B 0,C 180,E1 -10765.418,E2 -10765.418} C_VEL
LIN {X 0,Y 513.906,Z 357.816,A -85,B 0,C 180,E1 -10765.709,E2 -10765.709} C_VEL
LIN {X 0,Y 513.8,Z 357.19,A -85,B 0,C 180,E1 -10765.777,E2 -10765.777} C_VEL
LIN {X 0,Y 513.76,Z 357.223,A -85,B 0,C 180,E1 -10769.124,E2 -10769.124} C_VEL
LIN {X 0,Y 513.755,Z 357.232,A -85,B 0,C 180,E1 -10772.657,E2 -10772.657} C_VEL
LIN {X 0,Y 513.806,Z 357.223,A -85,B 0,C 180,E1 -10776.001,E2 -10776.001} C_VEL
LIN {X 0,Y 513.757,Z 357.223,A -85,B 0,C 180,E1 -10779.255,E2 -10779.255} C_VEL
LIN {X 0,Y 513.752,Z 357.221,A -85,B 0,C 180,E1 -10782.793,E2 -10782.793} C_VEL
LIN {X 0,Y 513.808,Z 357.209,A -85,B 0,C 180,E1 -10786.151,E2 -10786.151} C_VEL
LIN {X 0,Y 513.762,Z 357.217,A -85,B 0,C 180,E1 -10789.572,E2 -10789.572} C_VEL
LIN {X 0,Y 513.751,Z 357.231,A -85,B 0,C 180,E1 -10793.069,E2 -10793.069} C_VEL
LIN {X 0,Y 513.795,Z 357.231,A -85,B 0,C 180,E1 -10796.43,E2 -10796.43} C_VEL
LIN {X 0,Y 513.765,Z 357.223,A -85,B 0,C 180,E1 -10799.777,E2 -10799.777} C_VEL
LIN {X 0,Y 513.747,Z 357.214,A -85,B 0,C 180,E1 -10803.236,E2 -10803.236} C_VEL
LIN {X 0,Y 513.8,Z 357.208,A -85,B 0,C 180,E1 -10806.593,E2 -10806.593} C_VEL
LIN {X 0,Y 513.766,Z 357.227,A -85,B 0,C 180,E1 -10809.975,E2 -10809.975} C_VEL
LIN {X 0,Y 513.749,Z 357.234,A -85,B 0,C 180,E1 -10813.392,E2 -10813.392} C_VEL
LIN {X 0,Y 513.8,Z 357.219,A -85,B 0,C 180,E1 -10816.739,E2 -10816.739} C_VEL
LIN {X 0,Y 513.766,Z 357.213,A -85,B 0,C 180,E1 -10820.15,E2 -10820.15} C_VEL
LIN {X 0,Y 513.747,Z 357.213,A -85,B 0,C 180,E1 -10823.553,E2 -10823.553} C_VEL
LIN {X 0,Y 513.802,Z 357.209,A -85,B 0,C 180,E1 -10826.839,E2 -10826.839} C_VEL
LIN {X 0,Y 513.757,Z 357.233,A -85,B 0,C 180,E1 -10830.141,E2 -10830.141} C_VEL
LIN {X 0,Y 513.751,Z 357.237,A -85,B 0,C 180,E1 -10833.689,E2 -10833.689} C_VEL
LIN {X 0,Y 513.769,Z 357.249,A -85,B 0,C 180,E1 -10834.393,E2 -10834.393} C_VEL
LIN {X 0,Y 515.024,Z 360.596,A -85,B 0,C 180,E1 -10835.077,E2 -10835.077} C_VEL
LIN {X 0,Y 516.063,Z 362.715,A -85,B 0,C 180,E1 -10835.539,E2 -10835.539} C_VEL
LIN {X 0,Y 520.001,Z 370.822,A -85,B 0,C 180,E1 -10837.193,E2 -10837.193} C_VEL
LIN {X 0,Y 531.178,Z 386.55,A -85,B 0,C 180,E1 -10839.13,E2 -10839.13} C_VEL
LIN {X 0,Y 540.135,Z 399.555,A -85,B 0,C 180,E1 -10840.577,E2 -10840.577} C_VEL
LIN {X 0,Y 552.8,Z 419.25,A -85,B 0,C 180,E1 -10842.499,E2 -10842.499} C_VEL
LIN {X 0,Y 565.093,Z 440.191,A -85,B 0,C 180,E1 -10844.252,E2 -10844.252} C_VEL
LIN {X 0,Y 565.446,Z 441.491,A -85,B 0,C 180,E1 -10844.313,E2 -10844.313} C_VEL
LIN {X 0,Y 557.158,Z 695.623,A -85,B 0,C 180,E1 -10847.949,E2 -10847.949} C_VEL
LIN {X 0,Y 554.816,Z 765.296,A -85,B 0,C 180,E1 -10848.964,E2 -10848.964} C_VEL
LIN {X 0,Y 552.972,Z 790.672,A -85,B 0,C 180,E1 -10849.493,E2 -10849.493} C_VEL
LIN {X 0,Y 550.894,Z 812.588,A -85,B 0,C 180,E1 -10850.106,E2 -10850.106} C_VEL
LIN {X 0,Y 547.983,Z 837.747,A -85,B 0,C 180,E1 -10851.015,E2 -10851.015} C_VEL
LIN {X 0,Y 545.336,Z 857.683,A -85,B 0,C 180,E1 -10851.904,E2 -10851.904} C_VEL
LIN {X 0,Y 541.848,Z 881.103,A -85,B 0,C 180,E1 -10853.149,E2 -10853.149} C_VEL
LIN {X 0,Y 538.631,Z 900.807,A -85,B 0,C 180,E1 -10854.399,E2 -10854.399} C_VEL
LIN {X 0,Y 535.089,Z 921.401,A -85,B 0,C 180,E1 -10855.903,E2 -10855.903} C_VEL
LIN {X 0,Y 531.48,Z 940.876,A -85,B 0,C 180,E1 -10857.576,E2 -10857.576} C_VEL
LIN {X 0,Y 528.088,Z 959.291,A -85,B 0,C 180,E1 -10859.381,E2 -10859.381} C_VEL
LIN {X 0,Y 524.731,Z 977.206,A -85,B 0,C 180,E1 -10861.426,E2 -10861.426} C_VEL
LIN {X 0,Y 521.856,Z 993.063,A -85,B 0,C 180,E1 -10863.485,E2 -10863.485} C_VEL
LIN {X 0,Y 519.193,Z 1008.334,A -85,B 0,C 180,E1 -10865.782,E2 -10865.782} C_VEL
LIN {X 0,Y 517.135,Z 1021.066,A -85,B 0,C 180,E1 -10867.969,E2 -10867.969} C_VEL
LIN {X 0,Y 515.222,Z 1034.319,A -85,B 0,C 180,E1 -10870.618,E2 -10870.618} C_VEL
LIN {X 0,Y 514.012,Z 1044.168,A -85,B 0,C 180,E1 -10872.918,E2 -10872.918} C_VEL
LIN {X 0,Y 512.969,Z 1054.477,A -85,B 0,C 180,E1 -10875.783,E2 -10875.783} C_VEL
LIN {X 0,Y 512.43,Z 1061.513,A -85,B 0,C 180,E1 -10878.177,E2 -10878.177} C_VEL
LIN {X 0,Y 512.08,Z 1067.948,A -85,B 0,C 180,E1 -10880.9,E2 -10880.9} C_VEL
LIN {X 0,Y 511.952,Z 1072.229,A -85,B 0,C 180,E1 -10883.383,E2 -10883.383} C_VEL
LIN {X 0,Y 511.923,Z 1074.977,A -85,B 0,C 180,E1 -10885.631,E2 -10885.631} C_VEL
LIN {X 0,Y 511.911,Z 1076.831,A -85,B 0,C 180,E1 -10888.321,E2 -10888.321} C_VEL
LIN {X 0,Y 511.918,Z 1077.019,A -85,B 0,C 180,E1 -10890.783,E2 -10890.783} C_VEL
LIN {X 0,Y 511.926,Z 1076.08,A -85,B 0,C 180,E1 -10893.023,E2 -10893.023} C_VEL
LIN {X 0,Y 511.944,Z 1073.538,A -85,B 0,C 180,E1 -10895.717,E2 -10895.717} C_VEL
LIN {X 0,Y 512.027,Z 1069.641,A -85,B 0,C 180,E1 -10898.196,E2 -10898.196} C_VEL
LIN {X 0,Y 512.24,Z 1064.67,A -85,B 0,C 180,E1 -10900.573,E2 -10900.573} C_VEL
LIN {X 0,Y 512.757,Z 1056.97,A -85,B 0,C 180,E1 -10903.418,E2 -10903.418} C_VEL
LIN {X 0,Y 513.441,Z 1049.328,A -85,B 0,C 180,E1 -10905.705,E2 -10905.705} C_VEL
LIN {X 0,Y 514.565,Z 1039.422,A -85,B 0,C 180,E1 -10908.231,E2 -10908.231} C_VEL
LIN {X 0,Y 516.04,Z 1028.059,A -85,B 0,C 180,E1 -10910.649,E2 -10910.649} C_VEL
LIN {X 0,Y 517.93,Z 1015.659,A -85,B 0,C 180,E1 -10912.953,E2 -10912.953} C_VEL
LIN {X 0,Y 520.264,Z 1001.259,A -85,B 0,C 180,E1 -10915.256,E2 -10915.256} C_VEL
LIN {X 0,Y 522.677,Z 987.346,A -85,B 0,C 180,E1 -10917.207,E2 -10917.207} C_VEL
LIN {X 0,Y 525.97,Z 968.915,A -85,B 0,C 180,E1 -10919.462,E2 -10919.462} C_VEL
LIN {X 0,Y 528.937,Z 952.57,A -85,B 0,C 180,E1 -10921.196,E2 -10921.196} C_VEL
LIN {X 0,Y 532.546,Z 932.518,A -85,B 0,C 180,E1 -10923.054,E2 -10923.054} C_VEL
LIN {X 0,Y 535.794,Z 913.573,A -85,B 0,C 180,E1 -10924.564,E2 -10924.564} C_VEL
LIN {X 0,Y 539.247,Z 892.861,A -85,B 0,C 180,E1 -10926,E2 -10926} C_VEL
LIN {X 0,Y 542.496,Z 871.184,A -85,B 0,C 180,E1 -10927.262,E2 -10927.262} C_VEL
LIN {X 0,Y 545.627,Z 848.934,A -85,B 0,C 180,E1 -10928.362,E2 -10928.362} C_VEL
LIN {X 0,Y 548.355,Z 825.903,A -85,B 0,C 180,E1 -10929.286,E2 -10929.286} C_VEL
LIN {X 0,Y 550.466,Z 805.612,A -85,B 0,C 180,E1 -10929.95,E2 -10929.95} C_VEL
LIN {X 0,Y 552.599,Z 780.143,A -85,B 0,C 180,E1 -10930.591,E2 -10930.591} C_VEL
LIN {X 0,Y 553.847,Z 757.956,A -85,B 0,C 180,E1 -10930.995,E2 -10930.995} C_VEL
LIN {X 0,Y 561.199,Z 515.922,A -85,B 0,C 180,E1 -10934.434,E2 -10934.434} C_VEL
LIN {X 0,Y 563.46,Z 439.96,A -85,B 0,C 180,E1 -10935.532,E2 -10935.532} C_VEL
LIN {X 0,Y 550.144,Z 416.988,A -85,B 0,C 180,E1 -10937.335,E2 -10937.335} C_VEL
LIN {X 0,Y 539.004,Z 399.185,A -85,B 0,C 180,E1 -10938.934,E2 -10938.934} C_VEL
LIN {X 0,Y 527.646,Z 382.254,A -85,B 0,C 180,E1 -10940.663,E2 -10940.663} C_VEL
LIN {X 0,Y 519.6,Z 370.515,A -85,B 0,C 180,E1 -10941.99,E2 -10941.99} C_VEL
LIN {X 0,Y 515.191,Z 360.907,A -85,B 0,C 180,E1 -10943.842,E2 -10943.842} C_VEL
LIN {X 0,Y 513.785,Z 357.398,A -85,B 0,C 180,E1 -10944.516,E2 -10944.516} C_VEL
LIN {X 0,Y 513.752,Z 357.228,A -85,B 0,C 180,E1 -10947.905,E2 -10947.905} C_VEL
LIN {X 0,Y 513.814,Z 357.225,A -85,B 0,C 180,E1 -10951.144,E2 -10951.144} C_VEL
LIN {X 0,Y 513.757,Z 357.232,A -85,B 0,C 180,E1 -10954.562,E2 -10954.562} C_VEL
LIN {X 0,Y 513.75,Z 357.226,A -85,B 0,C 180,E1 -10958.057,E2 -10958.057} C_VEL
LIN {X 0,Y 513.802,Z 357.204,A -85,B 0,C 180,E1 -10961.393,E2 -10961.393} C_VEL
LIN {X 0,Y 513.757,Z 357.217,A -85,B 0,C 180,E1 -10964.767,E2 -10964.767} C_VEL
LIN {X 0,Y 513.752,Z 357.234,A -85,B 0,C 180,E1 -10968.322,E2 -10968.322} C_VEL
LIN {X 0,Y 513.8,Z 357.211,A -85,B 0,C 180,E1 -10971.72,E2 -10971.72} C_VEL
LIN {X 0,Y 513.757,Z 357.21,A -85,B 0,C 180,E1 -10974.976,E2 -10974.976} C_VEL
LIN {X 0,Y 513.753,Z 357.234,A -85,B 0,C 180,E1 -10978.439,E2 -10978.439} C_VEL
LIN {X 0,Y 513.804,Z 357.204,A -85,B 0,C 180,E1 -10981.784,E2 -10981.784} C_VEL
LIN {X 0,Y 513.757,Z 357.214,A -85,B 0,C 180,E1 -10985.136,E2 -10985.136} C_VEL
LIN {X 0,Y 513.754,Z 357.235,A -85,B 0,C 180,E1 -10988.625,E2 -10988.625} C_VEL
LIN {X 0,Y 513.799,Z 357.204,A -85,B 0,C 180,E1 -10992.019,E2 -10992.019} C_VEL
LIN {X 0,Y 513.756,Z 357.217,A -85,B 0,C 180,E1 -10995.233,E2 -10995.233} C_VEL
LIN {X 0,Y 513.758,Z 357.234,A -85,B 0,C 180,E1 -10998.731,E2 -10998.731} C_VEL
LIN {X 0,Y 513.814,Z 357.213,A -85,B 0,C 180,E1 -11002.134,E2 -11002.134} C_VEL
LIN {X 0,Y 513.758,Z 357.208,A -85,B 0,C 180,E1 -11005.475,E2 -11005.475} C_VEL
LIN {X 0,Y 513.756,Z 357.214,A -85,B 0,C 180,E1 -11008.987,E2 -11008.987} C_VEL
LIN {X 0,Y 513.805,Z 357.216,A -85,B 0,C 180,E1 -11012.355,E2 -11012.355} C_VEL
LIN {X 0,Y 513.769,Z 357.226,A -85,B 0,C 180,E1 -11015.751,E2 -11015.751} C_VEL
LIN {X 0,Y 513.753,Z 357.226,A -85,B 0,C 180,E1 -11019.237,E2 -11019.237} C_VEL
LIN {X 0,Y 513.784,Z 357.462,A -85,B 0,C 180,E1 -11019.356,E2 -11019.356} C_VEL
LIN {X 0,Y 514.977,Z 360.579,A -85,B 0,C 180,E1 -11019.594,E2 -11019.594} C_VEL
LIN {X 0,Y 517.692,Z 363.139,A -85,B 0,C 180,E1 -11020.029,E2 -11020.029} C_VEL
LIN {X 0,Y 520.579,Z 367.545,A -85,B 0,C 180,E1 -11020.518,E2 -11020.518} C_VEL
LIN {X 0,Y 522.439,Z 369.688,A -85,B 0,C 180,E1 -11020.813,E2 -11020.813} C_VEL
LIN {X 0,Y 525.872,Z 374.053,A -85,B 0,C 180,E1 -11021.356,E2 -11021.356} C_VEL
LIN {X 0,Y 538.036,Z 390.725,A -85,B 0,C 180,E1 -11023.204,E2 -11023.204} C_VEL
LIN {X 0,Y 547.707,Z 404.638,A -85,B 0,C 180,E1 -11024.583,E2 -11024.583} C_VEL
LIN {X 0,Y 561.292,Z 426.823,A -85,B 0,C 180,E1 -11026.435,E2 -11026.435} C_VEL
LIN {X 0,Y 563.671,Z 431.223,A -85,B 0,C 180,E1 -11026.753,E2 -11026.753} C_VEL
LIN {X 0,Y 556.034,Z 677.254,A -85,B 0,C 180,E1 -11030.249,E2 -11030.249} C_VEL
LIN {X 0,Y 553.889,Z 743.237,A -85,B 0,C 180,E1 -11031.206,E2 -11031.206} C_VEL
LIN {X 0,Y 552.273,Z 768.004,A -85,B 0,C 180,E1 -11031.735,E2 -11031.735} C_VEL
LIN {X 0,Y 550.403,Z 789.611,A -85,B 0,C 180,E1 -11032.348,E2 -11032.348} C_VEL
LIN {X 0,Y 547.847,Z 813.786,A -85,B 0,C 180,E1 -11033.227,E2 -11033.227} C_VEL
LIN {X 0,Y 546.087,Z 828.142,A -85,B 0,C 180,E1 -11033.849,E2 -11033.849} C_VEL
LIN {X 0,Y 544.328,Z 835.328,A -85,B 0,C 180,E1 -11034.127,E2 -11034.127} C_VEL
LIN {X 0,Y 536.947,Z 853.249,A -85,B 0,C 180,E1 -11034.68,E2 -11034.68} C_VEL
LIN {X 0,Y 535.072,Z 860.018,A -85,B 0,C 180,E1 -11035.016,E2 -11035.016} C_VEL
LIN {X 0,Y 531.924,Z 879.096,A -85,B 0,C 180,E1 -11036.257,E2 -11036.257} C_VEL
LIN {X 0,Y 528.155,Z 900.295,A -85,B 0,C 180,E1 -11037.861,E2 -11037.861} C_VEL
LIN {X 0,Y 524.745,Z 918.416,A -85,B 0,C 180,E1 -11039.461,E2 -11039.461} C_VEL
LIN {X 0,Y 521.189,Z 936.989,A -85,B 0,C 180,E1 -11041.339,E2 -11041.339} C_VEL
LIN {X 0,Y 517.932,Z 953.396,A -85,B 0,C 180,E1 -11043.268,E2 -11043.268} C_VEL
LIN {X 0,Y 514.808,Z 969.645,A -85,B 0,C 180,E1 -11045.44,E2 -11045.44} C_VEL
LIN {X 0,Y 512.011,Z 984.313,A -85,B 0,C 180,E1 -11047.737,E2 -11047.737} C_VEL
LIN {X 0,Y 509.654,Z 997.84,A -85,B 0,C 180,E1 -11050.159,E2 -11050.159} C_VEL
LIN {X 0,Y 507.692,Z 1009.794,A -85,B 0,C 180,E1 -11052.699,E2 -11052.699} C_VEL
LIN {X 0,Y 506.265,Z 1020.096,A -85,B 0,C 180,E1 -11055.24,E2 -11055.24} C_VEL
LIN {X 0,Y 505.212,Z 1028.916,A -85,B 0,C 180,E1 -11057.89,E2 -11057.89} C_VEL
LIN {X 0,Y 504.592,Z 1035.595,A -85,B 0,C 180,E1 -11060.303,E2 -11060.303} C_VEL
LIN {X 0,Y 504.172,Z 1041.795,A -85,B 0,C 180,E1 -11063.166,E2 -11063.166} C_VEL
LIN {X 0,Y 504.013,Z 1045.614,A -85,B 0,C 180,E1 -11065.563,E2 -11065.563} C_VEL
LIN {X 0,Y 503.947,Z 1048.597,A -85,B 0,C 180,E1 -11068.295,E2 -11068.295} C_VEL
LIN {X 0,Y 503.93,Z 1049.839,A -85,B 0,C 180,E1 -11070.91,E2 -11070.91} C_VEL
LIN {X 0,Y 503.926,Z 1049.843,A -85,B 0,C 180,E1 -11073.185,E2 -11073.185} C_VEL
LIN {X 0,Y 503.953,Z 1048.504,A -85,B 0,C 180,E1 -11075.922,E2 -11075.922} C_VEL
LIN {X 0,Y 504.014,Z 1045.603,A -85,B 0,C 180,E1 -11078.557,E2 -11078.557} C_VEL
LIN {X 0,Y 504.178,Z 1041.742,A -85,B 0,C 180,E1 -11080.98,E2 -11080.98} C_VEL
LIN {X 0,Y 504.618,Z 1035.46,A -85,B 0,C 180,E1 -11083.872,E2 -11083.872} C_VEL
LIN {X 0,Y 505.228,Z 1029.033,A -85,B 0,C 180,E1 -11086.204,E2 -11086.204} C_VEL
LIN {X 0,Y 506.311,Z 1020.118,A -85,B 0,C 180,E1 -11088.898,E2 -11088.898} C_VEL
LIN {X 0,Y 507.714,Z 1010.182,A -85,B 0,C 180,E1 -11091.367,E2 -11091.367} C_VEL
LIN {X 0,Y 509.527,Z 999.254,A -85,B 0,C 180,E1 -11093.721,E2 -11093.721} C_VEL
LIN {X 0,Y 511.928,Z 985.82,A -85,B 0,C 180,E1 -11096.195,E2 -11096.195} C_VEL
LIN {X 0,Y 514.478,Z 972.616,A -85,B 0,C 180,E1 -11098.308,E2 -11098.308} C_VEL
LIN {X 0,Y 517.843,Z 955.761,A -85,B 0,C 180,E1 -11100.647,E2 -11100.647} C_VEL
LIN {X 0,Y 520.978,Z 940.319,A -85,B 0,C 180,E1 -11102.506,E2 -11102.506} C_VEL
LIN {X 0,Y 524.868,Z 921.068,A -85,B 0,C 180,E1 -11104.524,E2 -11104.524} C_VEL
LIN {X 0,Y 528.307,Z 903.339,A -85,B 0,C 180,E1 -11106.125,E2 -11106.125} C_VEL
LIN {X 0,Y 532.095,Z 883.218,A -85,B 0,C 180,E1 -11107.709,E2 -11107.709} C_VEL
LIN {X 0,Y 535.572,Z 862.977,A -85,B 0,C 180,E1 -11109.057,E2 -11109.057} C_VEL
LIN {X 0,Y 538.989,Z 841.653,A -85,B 0,C 180,E1 -11110.279,E2 -11110.279} C_VEL
LIN {X 0,Y 542.071,Z 819.471,A -85,B 0,C 180,E1 -11111.327,E2 -11111.327} C_VEL
LIN {X 0,Y 544.441,Z 799.917,A -85,B 0,C 180,E1 -11112.101,E2 -11112.101} C_VEL
LIN {X 0,Y 546.964,Z 775.211,A -85,B 0,C 180,E1 -11112.883,E2 -11112.883} C_VEL
LIN {X 0,Y 548.613,Z 753.902,A -85,B 0,C 180,E1 -11113.392,E2 -11113.392} C_VEL
LIN {X 0,Y 549.906,Z 729.728,A -85,B 0,C 180,E1 -11113.82,E2 -11113.82} C_VEL
LIN {X 0,Y 558.448,Z 476.825,A -85,B 0,C 180,E1 -11117.46,E2 -11117.46} C_VEL
LIN {X 0,Y 559.794,Z 434.861,A -85,B 0,C 180,E1 -11118.085,E2 -11118.085} C_VEL
LIN {X 0,Y 548.365,Z 416.204,A -85,B 0,C 180,E1 -11119.746,E2 -11119.746} C_VEL
LIN {X 0,Y 539.659,Z 403.371,A -85,B 0,C 180,E1 -11121.072,E2 -11121.072} C_VEL
LIN {X 0,Y 530.243,Z 390.539,A -85,B 0,C 180,E1 -11122.578,E2 -11122.578} C_VEL
LIN {X 0,Y 522.245,Z 380.137,A -85,B 0,C 180,E1 -11123.932,E2 -11123.932} C_VEL
LIN {X 0,Y 518.411,Z 375.142,A -85,B 0,C 180,E1 -11124.612,E2 -11124.612} C_VEL
LIN {X 0,Y 515.16,Z 370.904,A -85,B 0,C 180,E1 -11125.205,E2 -11125.205} C_VEL
LIN {X 0,Y 511.277,Z 366.368,A -85,B 0,C 180,E1 -11125.923,E2 -11125.923} C_VEL
LIN {X 0,Y 510.058,Z 364.29,A -85,B 0,C 180,E1 -11126.169,E2 -11126.169} C_VEL
LIN {X 0,Y 507.318,Z 361.986,A -85,B 0,C 180,E1 -11126.674,E2 -11126.674} C_VEL
LIN {X 0,Y 505.948,Z 358.981,A -85,B 0,C 180,E1 -11126.977,E2 -11126.977} C_VEL
LIN {X 0,Y 505.819,Z 358.226,A -85,B 0,C 180,E1 -11127.023,E2 -11127.023} C_VEL
LIN {X 0,Y 505.821,Z 358.219,A -85,B 0,C 180,E1 -11130.514,E2 -11130.514} C_VEL
LIN {X 0,Y 505.867,Z 358.21,A -85,B 0,C 180,E1 -11133.846,E2 -11133.846} C_VEL
LIN {X 0,Y 505.817,Z 358.219,A -85,B 0,C 180,E1 -11137.204,E2 -11137.204} C_VEL
LIN {X 0,Y 505.818,Z 358.222,A -85,B 0,C 180,E1 -11140.724,E2 -11140.724} C_VEL
LIN {X 0,Y 505.867,Z 358.218,A -85,B 0,C 180,E1 -11144.171,E2 -11144.171} C_VEL
LIN {X 0,Y 505.827,Z 358.218,A -85,B 0,C 180,E1 -11147.557,E2 -11147.557} C_VEL
LIN {X 0,Y 505.81,Z 358.211,A -85,B 0,C 180,E1 -11151.015,E2 -11151.015} C_VEL
LIN {X 0,Y 505.861,Z 358.197,A -85,B 0,C 180,E1 -11154.328,E2 -11154.328} C_VEL
LIN {X 0,Y 505.825,Z 358.208,A -85,B 0,C 180,E1 -11157.734,E2 -11157.734} C_VEL
LIN {X 0,Y 505.814,Z 358.223,A -85,B 0,C 180,E1 -11161.133,E2 -11161.133} C_VEL
LIN {X 0,Y 505.86,Z 358.216,A -85,B 0,C 180,E1 -11164.535,E2 -11164.535} C_VEL
LIN {X 0,Y 505.819,Z 358.203,A -85,B 0,C 180,E1 -11167.839,E2 -11167.839} C_VEL
LIN {X 0,Y 505.809,Z 358.199,A -85,B 0,C 180,E1 -11171.334,E2 -11171.334} C_VEL
LIN {X 0,Y 505.856,Z 358.198,A -85,B 0,C 180,E1 -11174.773,E2 -11174.773} C_VEL
LIN {X 0,Y 505.836,Z 358.211,A -85,B 0,C 180,E1 -11178.199,E2 -11178.199} C_VEL
LIN {X 0,Y 505.811,Z 358.223,A -85,B 0,C 180,E1 -11181.573,E2 -11181.573} C_VEL
LIN {X 0,Y 505.86,Z 358.216,A -85,B 0,C 180,E1 -11184.899,E2 -11184.899} C_VEL
LIN {X 0,Y 505.833,Z 358.216,A -85,B 0,C 180,E1 -11188.321,E2 -11188.321} C_VEL
LIN {X 0,Y 505.809,Z 358.224,A -85,B 0,C 180,E1 -11191.785,E2 -11191.785} C_VEL
LIN {X 0,Y 505.856,Z 358.329,A -85,B 0,C 180,E1 -11193.236,E2 -11193.236} C_VEL
LIN {X 0,Y 507.026,Z 361.574,A -85,B 0,C 180,E1 -11193.924,E2 -11193.924} C_VEL
LIN {X 0,Y 508.127,Z 363.457,A -85,B 0,C 180,E1 -11194.386,E2 -11194.386} C_VEL
LIN {X 0,Y 511.472,Z 370.526,A -85,B 0,C 180,E1 -11195.873,E2 -11195.873} C_VEL
LIN {X 0,Y 517.191,Z 378.321,A -85,B 0,C 180,E1 -11196.943,E2 -11196.943} C_VEL
LIN {X 0,Y 526.687,Z 391.502,A -85,B 0,C 180,E1 -11198.618,E2 -11198.618} C_VEL
LIN {X 0,Y 538.736,Z 409.397,A -85,B 0,C 180,E1 -11200.599,E2 -11200.599} C_VEL
LIN {X 0,Y 550.421,Z 428.049,A -85,B 0,C 180,E1 -11202.391,E2 -11202.391} C_VEL
LIN {X 0,Y 559.833,Z 444.357,A -85,B 0,C 180,E1 -11203.761,E2 -11203.761} C_VEL
LIN {X 0,Y 551.218,Z 697.847,A -85,B 0,C 180,E1 -11207.416,E2 -11207.416} C_VEL
LIN {X 0,Y 548.851,Z 765.211,A -85,B 0,C 180,E1 -11208.406,E2 -11208.406} C_VEL
LIN {X 0,Y 546.947,Z 790.534,A -85,B 0,C 180,E1 -11208.938,E2 -11208.938} C_VEL
LIN {X 0,Y 544.812,Z 812.3,A -85,B 0,C 180,E1 -11209.551,E2 -11209.551} C_VEL
LIN {X 0,Y 541.812,Z 837.253,A -85,B 0,C 180,E1 -11210.455,E2 -11210.455} C_VEL
LIN {X 0,Y 538.992,Z 857.715,A -85,B 0,C 180,E1 -11211.373,E2 -11211.373} C_VEL
LIN {X 0,Y 535.358,Z 881.083,A -85,B 0,C 180,E1 -11212.627,E2 -11212.627} C_VEL
LIN {X 0,Y 532.124,Z 900.104,A -85,B 0,C 180,E1 -11213.841,E2 -11213.841} C_VEL
LIN {X 0,Y 528.453,Z 920.63,A -85,B 0,C 180,E1 -11215.349,E2 -11215.349} C_VEL
LIN {X 0,Y 524.681,Z 940.175,A -85,B 0,C 180,E1 -11217.038,E2 -11217.038} C_VEL
LIN {X 0,Y 521.204,Z 958.071,A -85,B 0,C 180,E1 -11218.804,E2 -11218.804} C_VEL
LIN {X 0,Y 517.662,Z 976.147,A -85,B 0,C 180,E1 -11220.873,E2 -11220.873} C_VEL
LIN {X 0,Y 514.766,Z 991.223,A -85,B 0,C 180,E1 -11222.841,E2 -11222.841} C_VEL
LIN {X 0,Y 511.753,Z 1007.595,A -85,B 0,C 180,E1 -11225.305,E2 -11225.305} C_VEL
LIN {X 0,Y 509.578,Z 1020.26,A -85,B 0,C 180,E1 -11227.503,E2 -11227.503} C_VEL
LIN {X 0,Y 507.526,Z 1033.62,A -85,B 0,C 180,E1 -11230.192,E2 -11230.192} C_VEL
LIN {X 0,Y 506.184,Z 1043.698,A -85,B 0,C 180,E1 -11232.573,E2 -11232.573} C_VEL
LIN {X 0,Y 505.112,Z 1053.565,A -85,B 0,C 180,E1 -11235.322,E2 -11235.322} C_VEL
LIN {X 0,Y 504.506,Z 1060.698,A -85,B 0,C 180,E1 -11237.757,E2 -11237.757} C_VEL
LIN {X 0,Y 504.146,Z 1066.814,A -85,B 0,C 180,E1 -11240.307,E2 -11240.307} C_VEL
LIN {X 0,Y 503.971,Z 1071.694,A -85,B 0,C 180,E1 -11243.049,E2 -11243.049} C_VEL
LIN {X 0,Y 503.931,Z 1074.534,A -85,B 0,C 180,E1 -11245.334,E2 -11245.334} C_VEL
LIN {X 0,Y 503.925,Z 1076.418,A -85,B 0,C 180,E1 -11247.839,E2 -11247.839} C_VEL
LIN {X 0,Y 503.916,Z 1076.851,A -85,B 0,C 180,E1 -11250.568,E2 -11250.568} C_VEL
LIN {X 0,Y 503.926,Z 1076.004,A -85,B 0,C 180,E1 -11252.843,E2 -11252.843} C_VEL
LIN {X 0,Y 503.939,Z 1073.839,A -85,B 0,C 180,E1 -11255.351,E2 -11255.351} C_VEL
LIN {X 0,Y 504.022,Z 1069.764,A -85,B 0,C 180,E1 -11258.137,E2 -11258.137} C_VEL
LIN {X 0,Y 504.23,Z 1064.959,A -85,B 0,C 180,E1 -11260.512,E2 -11260.512} C_VEL
LIN {X 0,Y 504.701,Z 1058.167,A -85,B 0,C 180,E1 -11263.169,E2 -11263.169} C_VEL
LIN {X 0,Y 505.456,Z 1049.904,A -85,B 0,C 180,E1 -11265.724,E2 -11265.724} C_VEL
LIN {X 0,Y 506.477,Z 1041.045,A -85,B 0,C 180,E1 -11268.056,E2 -11268.056} C_VEL
LIN {X 0,Y 508.133,Z 1028.955,A -85,B 0,C 180,E1 -11270.744,E2 -11270.744} C_VEL
LIN {X 0,Y 509.968,Z 1017.316,A -85,B 0,C 180,E1 -11272.966,E2 -11272.966} C_VEL
LIN {X 0,Y 512.628,Z 1001.746,A -85,B 0,C 180,E1 -11275.535,E2 -11275.535} C_VEL
LIN {X 0,Y 515.141,Z 987.899,A -85,B 0,C 180,E1 -11277.514,E2 -11277.514} C_VEL
LIN {X 0,Y 518.363,Z 970.778,A -85,B 0,C 180,E1 -11279.667,E2 -11279.667} C_VEL
LIN {X 0,Y 521.652,Z 953.358,A -85,B 0,C 180,E1 -11281.552,E2 -11281.552} C_VEL
LIN {X 0,Y 525.288,Z 934.182,A -85,B 0,C 180,E1 -11283.375,E2 -11283.375} C_VEL
LIN {X 0,Y 528.894,Z 913.938,A -85,B 0,C 180,E1 -11285.014,E2 -11285.014} C_VEL
LIN {X 0,Y 532.482,Z 893.313,A -85,B 0,C 180,E1 -11286.464,E2 -11286.464} C_VEL
LIN {X 0,Y 535.856,Z 871.76,A -85,B 0,C 180,E1 -11287.737,E2 -11287.737} C_VEL
LIN {X 0,Y 539.01,Z 850.159,A -85,B 0,C 180,E1 -11288.819,E2 -11288.819} C_VEL
LIN {X 0,Y 541.922,Z 826.849,A -85,B 0,C 180,E1 -11289.776,E2 -11289.776} C_VEL
LIN {X 0,Y 544.113,Z 806.615,A -85,B 0,C 180,E1 -11290.449,E2 -11290.449} C_VEL
LIN {X 0,Y 546.315,Z 781.962,A -85,B 0,C 180,E1 -11291.089,E2 -11291.089} C_VEL
LIN {X 0,Y 547.686,Z 758.897,A -85,B 0,C 180,E1 -11291.519,E2 -11291.519} C_VEL
LIN {X 0,Y 555.231,Z 521.007,A -85,B 0,C 180,E1 -11294.93,E2 -11294.93} C_VEL
LIN {X 0,Y 557.675,Z 443.181,A -85,B 0,C 180,E1 -11296.062,E2 -11296.062} C_VEL
LIN {X 0,Y 544.63,Z 420.749,A -85,B 0,C 180,E1 -11297.875,E2 -11297.875} C_VEL
LIN {X 0,Y 532.554,Z 401.419,A -85,B 0,C 180,E1 -11299.662,E2 -11299.662} C_VEL
LIN {X 0,Y 522.976,Z 387.268,A -85,B 0,C 180,E1 -11301.162,E2 -11301.162} C_VEL
LIN {X 0,Y 514.362,Z 375.002,A -85,B 0,C 180,E1 -11302.592,E2 -11302.592} C_VEL
LIN {X 0,Y 511.191,Z 370.226,A -85,B 0,C 180,E1 -11303.165,E2 -11303.165} C_VEL
LIN {X 0,Y 507.157,Z 361.687,A -85,B 0,C 180,E1 -11304.905,E2 -11304.905} C_VEL
LIN {X 0,Y 505.824,Z 358.204,A -85,B 0,C 180,E1 -11305.642,E2 -11305.642} C_VEL
LIN {X 0,Y 505.852,Z 358.197,A -85,B 0,C 180,E1 -11308.942,E2 -11308.942} C_VEL
LIN {X 0,Y 505.811,Z 358.2,A -85,B 0,C 180,E1 -11312.326,E2 -11312.326} C_VEL
LIN {X 0,Y 505.823,Z 358.203,A -85,B 0,C 180,E1 -11315.846,E2 -11315.846} C_VEL
LIN {X 0,Y 505.861,Z 358.219,A -85,B 0,C 180,E1 -11319.158,E2 -11319.158} C_VEL
LIN {X 0,Y 505.814,Z 358.22,A -85,B 0,C 180,E1 -11322.633,E2 -11322.633} C_VEL
LIN {X 0,Y 505.814,Z 358.199,A -85,B 0,C 180,E1 -11326.161,E2 -11326.161} C_VEL
LIN {X 0,Y 505.862,Z 358.197,A -85,B 0,C 180,E1 -11329.523,E2 -11329.523} C_VEL
LIN {X 0,Y 505.823,Z 358.222,A -85,B 0,C 180,E1 -11332.96,E2 -11332.96} C_VEL
LIN {X 0,Y 505.81,Z 358.202,A -85,B 0,C 180,E1 -11336.487,E2 -11336.487} C_VEL
LIN {X 0,Y 505.858,Z 358.193,A -85,B 0,C 180,E1 -11339.887,E2 -11339.887} C_VEL
LIN {X 0,Y 505.833,Z 358.221,A -85,B 0,C 180,E1 -11343.286,E2 -11343.286} C_VEL
LIN {X 0,Y 505.808,Z 358.199,A -85,B 0,C 180,E1 -11346.698,E2 -11346.698} C_VEL
LIN {X 0,Y 505.858,Z 358.198,A -85,B 0,C 180,E1 -11350.017,E2 -11350.017} C_VEL
LIN {X 0,Y 505.837,Z 358.22,A -85,B 0,C 180,E1 -11353.489,E2 -11353.489} C_VEL
LIN {X 0,Y 505.811,Z 358.202,A -85,B 0,C 180,E1 -11356.908,E2 -11356.908} C_VEL
LIN {X 0,Y 505.858,Z 358.195,A -85,B 0,C 180,E1 -11360.237,E2 -11360.237} C_VEL
LIN {X 0,Y 505.829,Z 358.223,A -85,B 0,C 180,E1 -11363.535,E2 -11363.535} C_VEL
LIN {X 0,Y 505.815,Z 358.223,A -85,B 0,C 180,E1 -11367.043,E2 -11367.043} C_VEL
LIN {X 0,Y 505.863,Z 358.201,A -85,B 0,C 180,E1 -11370.399,E2 -11370.399} C_VEL
LIN {X 0,Y 505.831,Z 358.202,A -85,B 0,C 180,E1 -11373.743,E2 -11373.743} C_VEL
LIN {X 0,Y 505.814,Z 358.208,A -85,B 0,C 180,E1 -11377.222,E2 -11377.222} C_VEL
LIN {X 0,Y 505.887,Z 358.359,A -85,B 0,C 180,E1 -11378.218,E2 -11378.218} C_VEL
LIN {X 0,Y 507.038,Z 361.49,A -85,B 0,C 180,E1 -11378.463,E2 -11378.463} C_VEL
LIN {X 0,Y 509.577,Z 364.042,A -85,B 0,C 180,E1 -11378.896,E2 -11378.896} C_VEL
LIN {X 0,Y 510.514,Z 365.429,A -85,B 0,C 180,E1 -11379.064,E2 -11379.064} C_VEL
LIN {X 0,Y 513.243,Z 369.092,A -85,B 0,C 180,E1 -11379.537,E2 -11379.537} C_VEL
LIN {X 0,Y 514.716,Z 370.731,A -85,B 0,C 180,E1 -11379.781,E2 -11379.781} C_VEL
LIN {X 0,Y 517.989,Z 375.01,A -85,B 0,C 180,E1 -11380.327,E2 -11380.327} C_VEL
LIN {X 0,Y 531.008,Z 392.505,A -85,B 0,C 180,E1 -11382.386,E2 -11382.386} C_VEL
LIN {X 0,Y 543.149,Z 409.924,A -85,B 0,C 180,E1 -11384.17,E2 -11384.17} C_VEL
LIN {X 0,Y 556.689,Z 432.23,A -85,B 0,C 180,E1 -11386.057,E2 -11386.057} C_VEL
LIN {X 0,Y 557.876,Z 434.704,A -85,B 0,C 180,E1 -11386.225,E2 -11386.225} C_VEL
LIN {X 0,Y 549.927,Z 680.362,A -85,B 0,C 180,E1 -11389.744,E2 -11389.744} C_VEL
LIN {X 0,Y 547.775,Z 743.673,A -85,B 0,C 180,E1 -11390.671,E2 -11390.671} C_VEL
LIN {X 0,Y 546.096,Z 768.42,A -85,B 0,C 180,E1 -11391.205,E2 -11391.205} C_VEL
LIN {X 0,Y 544.147,Z 790.154,A -85,B 0,C 180,E1 -11391.828,E2 -11391.828} C_VEL
LIN {X 0,Y 541.471,Z 814.447,A -85,B 0,C 180,E1 -11392.721,E2 -11392.721} C_VEL
LIN {X 0,Y 538.798,Z 834.992,A -85,B 0,C 180,E1 -11393.65,E2 -11393.65} C_VEL
LIN {X 0,Y 535.419,Z 857.913,A -85,B 0,C 180,E1 -11394.887,E2 -11394.887} C_VEL
LIN {X 0,Y 535.072,Z 860.018,A -85,B 0,C 180,E1 -11395.016,E2 -11395.016} C_VEL
LIN {X 0,Y 533.151,Z 866.91,A -85,B 0,C 180,E1 -11395.373,E2 -11395.373} C_VEL
LIN {X 0,Y 525.296,Z 883.992,A -85,B 0,C 180,E1 -11396.14,E2 -11396.14} C_VEL
LIN {X 0,Y 523.292,Z 890.316,A -85,B 0,C 180,E1 -11396.56,E2 -11396.56} C_VEL
LIN {X 0,Y 519.831,Z 908.643,A -85,B 0,C 180,E1 -11398.065,E2 -11398.065} C_VEL
LIN {X 0,Y 515.922,Z 928.193,A -85,B 0,C 180,E1 -11399.931,E2 -11399.931} C_VEL
LIN {X 0,Y 512.604,Z 944.372,A -85,B 0,C 180,E1 -11401.706,E2 -11401.706} C_VEL
LIN {X 0,Y 508.891,Z 962.559,A -85,B 0,C 180,E1 -11404.014,E2 -11404.014} C_VEL
LIN {X 0,Y 506.164,Z 976.066,A -85,B 0,C 180,E1 -11405.987,E2 -11405.987} C_VEL
LIN {X 0,Y 503.35,Z 990.707,A -85,B 0,C 180,E1 -11408.439,E2 -11408.439} C_VEL
LIN {X 0,Y 501.164,Z 1002.678,A -85,B 0,C 180,E1 -11410.78,E2 -11410.78} C_VEL
LIN {X 0,Y 499.344,Z 1014.112,A -85,B 0,C 180,E1 -11413.361,E2 -11413.361} C_VEL
LIN {X 0,Y 497.986,Z 1023.606,A -85,B 0,C 180,E1 -11415.939,E2 -11415.939} C_VEL
LIN {X 0,Y 497.066,Z 1031.627,A -85,B 0,C 180,E1 -11418.513,E2 -11418.513} C_VEL
LIN {X 0,Y 496.434,Z 1038.548,A -85,B 0,C 180,E1 -11421.312,E2 -11421.312} C_VEL
LIN {X 0,Y 496.146,Z 1043.064,A -85,B 0,C 180,E1 -11423.636,E2 -11423.636} C_VEL
LIN {X 0,Y 495.985,Z 1047.067,A -85,B 0,C 180,E1 -11426.417,E2 -11426.417} C_VEL
LIN {X 0,Y 495.938,Z 1049.294,A -85,B 0,C 180,E1 -11429.076,E2 -11429.076} C_VEL
LIN {X 0,Y 495.918,Z 1050.148,A -85,B 0,C 180,E1 -11431.386,E2 -11431.386} C_VEL
LIN {X 0,Y 495.936,Z 1049.805,A -85,B 0,C 180,E1 -11434.162,E2 -11434.162} C_VEL
LIN {X 0,Y 495.968,Z 1048.022,A -85,B 0,C 180,E1 -11436.715,E2 -11436.715} C_VEL
LIN {X 0,Y 496.06,Z 1045.155,A -85,B 0,C 180,E1 -11439.163,E2 -11439.163} C_VEL
LIN {X 0,Y 496.332,Z 1040.111,A -85,B 0,C 180,E1 -11442.094,E2 -11442.094} C_VEL
LIN {X 0,Y 496.805,Z 1034.416,A -85,B 0,C 180,E1 -11444.571,E2 -11444.571} C_VEL
LIN {X 0,Y 497.664,Z 1026.716,A -85,B 0,C 180,E1 -11447.299,E2 -11447.299} C_VEL
LIN {X 0,Y 498.91,Z 1017.376,A -85,B 0,C 180,E1 -11449.957,E2 -11449.957} C_VEL
LIN {X 0,Y 500.649,Z 1006.723,A -85,B 0,C 180,E1 -11452.548,E2 -11452.548} C_VEL
LIN {X 0,Y 502.833,Z 994.441,A -85,B 0,C 180,E1 -11455.059,E2 -11455.059} C_VEL
LIN {X 0,Y 505.349,Z 981.711,A -85,B 0,C 180,E1 -11457.327,E2 -11457.327} C_VEL
LIN {X 0,Y 508.518,Z 966.224,A -85,B 0,C 180,E1 -11459.703,E2 -11459.703} C_VEL
LIN {X 0,Y 511.718,Z 951.187,A -85,B 0,C 180,E1 -11461.71,E2 -11461.71} C_VEL
LIN {X 0,Y 515.692,Z 932.365,A -85,B 0,C 180,E1 -11463.886,E2 -11463.886} C_VEL
LIN {X 0,Y 519.195,Z 915.589,A -85,B 0,C 180,E1 -11465.564,E2 -11465.564} C_VEL
LIN {X 0,Y 523.484,Z 894.286,A -85,B 0,C 180,E1 -11467.402,E2 -11467.402} C_VEL
LIN {X 0,Y 526.959,Z 875.808,A -85,B 0,C 180,E1 -11468.768,E2 -11468.768} C_VEL
LIN {X 0,Y 530.668,Z 854.628,A -85,B 0,C 180,E1 -11470.121,E2 -11470.121} C_VEL
LIN {X 0,Y 533.938,Z 833.645,A -85,B 0,C 180,E1 -11471.237,E2 -11471.237} C_VEL
LIN {X 0,Y 537.103,Z 810.848,A -85,B 0,C 180,E1 -11472.262,E2 -11472.262} C_VEL
LIN {X 0,Y 539.796,Z 787.034,A -85,B 0,C 180,E1 -11473.105,E2 -11473.105} C_VEL
LIN {X 0,Y 542.027,Z 763.422,A -85,B 0,C 180,E1 -11473.761,E2 -11473.761} C_VEL
LIN {X 0,Y 543.601,Z 738.929,A -85,B 0,C 180,E1 -11474.245,E2 -11474.245} C_VEL
LIN {X 0,Y 552.114,Z 499.336,A -85,B 0,C 180,E1 -11477.736,E2 -11477.736} C_VEL
LIN {X 0,Y 554.239,Z 438.354,A -85,B 0,C 180,E1 -11478.64,E2 -11478.64} C_VEL
LIN {X 0,Y 541.092,Z 417.091,A -85,B 0,C 180,E1 -11480.615,E2 -11480.615} C_VEL
LIN {X 0,Y 530.106,Z 401.533,A -85,B 0,C 180,E1 -11482.363,E2 -11482.363} C_VEL
LIN {X 0,Y 519.296,Z 387.153,A -85,B 0,C 180,E1 -11484.207,E2 -11484.207} C_VEL
LIN {X 0,Y 514.694,Z 381.339,A -85,B 0,C 180,E1 -11485.034,E2 -11485.034} C_VEL
LIN {X 0,Y 510.833,Z 376.392,A -85,B 0,C 180,E1 -11485.754,E2 -11485.754} C_VEL
LIN {X 0,Y 507.61,Z 372.243,A -85,B 0,C 180,E1 -11486.374,E2 -11486.374} C_VEL
LIN {X 0,Y 506.536,Z 370.989,A -85,B 0,C 180,E1 -11486.582,E2 -11486.582} C_VEL
LIN {X 0,Y 503.64,Z 367.828,A -85,B 0,C 180,E1 -11487.146,E2 -11487.146} C_VEL
LIN {X 0,Y 502.365,Z 365.417,A -85,B 0,C 180,E1 -11487.425,E2 -11487.425} C_VEL
LIN {X 0,Y 499.464,Z 363.017,A -85,B 0,C 180,E1 -11487.994,E2 -11487.994} C_VEL
LIN {X 0,Y 498.07,Z 360.156,A -85,B 0,C 180,E1 -11488.317,E2 -11488.317} C_VEL
LIN {X 0,Y 497.886,Z 359.196,A -85,B 0,C 180,E1 -11488.388,E2 -11488.388} C_VEL
LIN {X 0,Y 497.942,Z 359.189,A -85,B 0,C 180,E1 -11491.828,E2 -11491.828} C_VEL
LIN {X 0,Y 497.886,Z 359.195,A -85,B 0,C 180,E1 -11495.309,E2 -11495.309} C_VEL
LIN {X 0,Y 497.874,Z 359.195,A -85,B 0,C 180,E1 -11498.808,E2 -11498.808} C_VEL
LIN {X 0,Y 497.913,Z 359.189,A -85,B 0,C 180,E1 -11502.227,E2 -11502.227} C_VEL
LIN {X 0,Y 497.889,Z 359.193,A -85,B 0,C 180,E1 -11505.58,E2 -11505.58} C_VEL
LIN {X 0,Y 497.873,Z 359.204,A -85,B 0,C 180,E1 -11509.001,E2 -11509.001} C_VEL
LIN {X 0,Y 497.92,Z 359.208,A -85,B 0,C 180,E1 -11512.384,E2 -11512.384} C_VEL
LIN {X 0,Y 497.899,Z 359.204,A -85,B 0,C 180,E1 -11515.854,E2 -11515.854} C_VEL
LIN {X 0,Y 497.869,Z 359.195,A -85,B 0,C 180,E1 -11519.31,E2 -11519.31} C_VEL
LIN {X 0,Y 497.905,Z 359.186,A -85,B 0,C 180,E1 -11522.647,E2 -11522.647} C_VEL
LIN {X 0,Y 497.906,Z 359.195,A -85,B 0,C 180,E1 -11526.11,E2 -11526.11} C_VEL
LIN {X 0,Y 497.871,Z 359.213,A -85,B 0,C 180,E1 -11529.479,E2 -11529.479} C_VEL
LIN {X 0,Y 497.892,Z 359.209,A -85,B 0,C 180,E1 -11532.998,E2 -11532.998} C_VEL
LIN {X 0,Y 497.908,Z 359.189,A -85,B 0,C 180,E1 -11536.329,E2 -11536.329} C_VEL
LIN {X 0,Y 497.868,Z 359.188,A -85,B 0,C 180,E1 -11539.719,E2 -11539.719} C_VEL
LIN {X 0,Y 497.89,Z 359.187,A -85,B 0,C 180,E1 -11543.18,E2 -11543.18} C_VEL
LIN {X 0,Y 497.924,Z 359.186,A -85,B 0,C 180,E1 -11546.669,E2 -11546.669} C_VEL
LIN {X 0,Y 497.876,Z 359.211,A -85,B 0,C 180,E1 -11550.051,E2 -11550.051} C_VEL
LIN {X 0,Y 497.886,Z 359.31,A -85,B 0,C 180,E1 -11551.977,E2 -11551.977} C_VEL
LIN {X 0,Y 499.189,Z 362.632,A -85,B 0,C 180,E1 -11552.74,E2 -11552.74} C_VEL
LIN {X 0,Y 500.218,Z 364.49,A -85,B 0,C 180,E1 -11553.21,E2 -11553.21} C_VEL
LIN {X 0,Y 502.776,Z 369.865,A -85,B 0,C 180,E1 -11554.423,E2 -11554.423} C_VEL
LIN {X 0,Y 513.514,Z 384.325,A -85,B 0,C 180,E1 -11556.52,E2 -11556.52} C_VEL
LIN {X 0,Y 523.228,Z 398.04,A -85,B 0,C 180,E1 -11558.273,E2 -11558.273} C_VEL
LIN {X 0,Y 534.82,Z 415.4,A -85,B 0,C 180,E1 -11560.219,E2 -11560.219} C_VEL
LIN {X 0,Y 546.385,Z 434.053,A -85,B 0,C 180,E1 -11562.031,E2 -11562.031} C_VEL
LIN {X 0,Y 554.244,Z 447.991,A -85,B 0,C 180,E1 -11563.208,E2 -11563.208} C_VEL
LIN {X 0,Y 545.342,Z 699.596,A -85,B 0,C 180,E1 -11566.865,E2 -11566.865} C_VEL
LIN {X 0,Y 542.94,Z 765.137,A -85,B 0,C 180,E1 -11567.837,E2 -11567.837} C_VEL
LIN {X 0,Y 540.977,Z 790.404,A -85,B 0,C 180,E1 -11568.372,E2 -11568.372} C_VEL
LIN {X 0,Y 538.79,Z 811.938,A -85,B 0,C 180,E1 -11568.98,E2 -11568.98} C_VEL
LIN {X 0,Y 535.62,Z 837.328,A -85,B 0,C 180,E1 -11569.906,E2 -11569.906} C_VEL
LIN {X 0,Y 532.72,Z 857.586,A -85,B 0,C 180,E1 -11570.822,E2 -11570.822} C_VEL
LIN {X 0,Y 528.916,Z 881.067,A -85,B 0,C 180,E1 -11572.092,E2 -11572.092} C_VEL
LIN {X 0,Y 525.437,Z 900.712,A -85,B 0,C 180,E1 -11573.361,E2 -11573.361} C_VEL
LIN {X 0,Y 521.595,Z 921.255,A -85,B 0,C 180,E1 -11574.894,E2 -11574.894} C_VEL
LIN {X 0,Y 517.677,Z 940.697,A -85,B 0,C 180,E1 -11576.6,E2 -11576.6} C_VEL
LIN {X 0,Y 513.853,Z 959.576,A -85,B 0,C 180,E1 -11578.496,E2 -11578.496} C_VEL
LIN {X 0,Y 510.258,Z 976.954,A -85,B 0,C 180,E1 -11580.537,E2 -11580.537} C_VEL
LIN {X 0,Y 506.928,Z 993.639,A -85,B 0,C 180,E1 -11582.767,E2 -11582.767} C_VEL
LIN {X 0,Y 503.991,Z 1008.732,A -85,B 0,C 180,E1 -11585.128,E2 -11585.128} C_VEL
LIN {X 0,Y 501.516,Z 1022.662,A -85,B 0,C 180,E1 -11587.617,E2 -11587.617} C_VEL
LIN {X 0,Y 499.522,Z 1035.008,A -85,B 0,C 180,E1 -11590.227,E2 -11590.227} C_VEL
LIN {X 0,Y 498.083,Z 1045.661,A -85,B 0,C 180,E1 -11592.837,E2 -11592.837} C_VEL
LIN {X 0,Y 497.047,Z 1054.808,A -85,B 0,C 180,E1 -11595.555,E2 -11595.555} C_VEL
LIN {X 0,Y 496.461,Z 1061.733,A -85,B 0,C 180,E1 -11598.027,E2 -11598.027} C_VEL
LIN {X 0,Y 496.072,Z 1068.23,A -85,B 0,C 180,E1 -11600.988,E2 -11600.988} C_VEL
LIN {X 0,Y 495.952,Z 1072.14,A -85,B 0,C 180,E1 -11603.401,E2 -11603.401} C_VEL
LIN {X 0,Y 495.92,Z 1075.135,A -85,B 0,C 180,E1 -11606.069,E2 -11606.069} C_VEL
LIN {X 0,Y 495.924,Z 1076.499,A -85,B 0,C 180,E1 -11608.729,E2 -11608.729} C_VEL
LIN {X 0,Y 495.93,Z 1076.545,A -85,B 0,C 180,E1 -11611.04,E2 -11611.04} C_VEL
LIN {X 0,Y 495.924,Z 1075.362,A -85,B 0,C 180,E1 -11613.595,E2 -11613.595} C_VEL
LIN {X 0,Y 495.952,Z 1072.445,A -85,B 0,C 180,E1 -11616.366,E2 -11616.366} C_VEL
LIN {X 0,Y 496.055,Z 1068.768,A -85,B 0,C 180,E1 -11618.695,E2 -11618.695} C_VEL
LIN {X 0,Y 496.357,Z 1063.169,A -85,B 0,C 180,E1 -11621.386,E2 -11621.386} C_VEL
LIN {X 0,Y 496.943,Z 1055.708,A -85,B 0,C 180,E1 -11624.11,E2 -11624.11} C_VEL
LIN {X 0,Y 497.799,Z 1047.592,A -85,B 0,C 180,E1 -11626.572,E2 -11626.572} C_VEL
LIN {X 0,Y 499.241,Z 1036.445,A -85,B 0,C 180,E1 -11629.381,E2 -11629.381} C_VEL
LIN {X 0,Y 500.875,Z 1025.768,A -85,B 0,C 180,E1 -11631.673,E2 -11631.673} C_VEL
LIN {X 0,Y 503.406,Z 1010.951,A -85,B 0,C 180,E1 -11634.402,E2 -11634.402} C_VEL
LIN {X 0,Y 505.876,Z 997.537,A -85,B 0,C 180,E1 -11636.532,E2 -11636.532} C_VEL
LIN {X 0,Y 509.269,Z 980.036,A -85,B 0,C 180,E1 -11638.945,E2 -11638.945} C_VEL
LIN {X 0,Y 512.399,Z 964.186,A -85,B 0,C 180,E1 -11640.838,E2 -11640.838} C_VEL
LIN {X 0,Y 516.202,Z 944.946,A -85,B 0,C 180,E1 -11642.845,E2 -11642.845} C_VEL
LIN {X 0,Y 519.647,Z 927.057,A -85,B 0,C 180,E1 -11644.451,E2 -11644.451} C_VEL
LIN {X 0,Y 523.461,Z 906.852,A -85,B 0,C 180,E1 -11646.038,E2 -11646.038} C_VEL
LIN {X 0,Y 527.087,Z 885.661,A -85,B 0,C 180,E1 -11647.444,E2 -11647.444} C_VEL
LIN {X 0,Y 530.399,Z 865.227,A -85,B 0,C 180,E1 -11648.608,E2 -11648.608} C_VEL
LIN {X 0,Y 533.687,Z 841.975,A -85,B 0,C 180,E1 -11649.708,E2 -11649.708} C_VEL
LIN {X 0,Y 536.297,Z 821.174,A -85,B 0,C 180,E1 -11650.518,E2 -11650.518} C_VEL
LIN {X 0,Y 539.015,Z 795.008,A -85,B 0,C 180,E1 -11651.32,E2 -11651.32} C_VEL
LIN {X 0,Y 540.806,Z 772.943,A -85,B 0,C 180,E1 -11651.822,E2 -11651.822} C_VEL
LIN {X 0,Y 542.31,Z 740.397,A -85,B 0,C 180,E1 -11652.349,E2 -11652.349} C_VEL
LIN {X 0,Y 550.562,Z 489.738,A -85,B 0,C 180,E1 -11655.961,E2 -11655.961} C_VEL
LIN {X 0,Y 551.919,Z 446.519,A -85,B 0,C 180,E1 -11656.603,E2 -11656.603} C_VEL
LIN {X 0,Y 538.465,Z 423.266,A -85,B 0,C 180,E1 -11658.53,E2 -11658.53} C_VEL
LIN {X 0,Y 525.532,Z 402.827,A -85,B 0,C 180,E1 -11660.509,E2 -11660.509} C_VEL
LIN {X 0,Y 514.351,Z 386.33,A -85,B 0,C 180,E1 -11662.345,E2 -11662.345} C_VEL
LIN {X 0,Y 506.757,Z 375.71,A -85,B 0,C 180,E1 -11663.67,E2 -11663.67} C_VEL
LIN {X 0,Y 502.476,Z 369.783,A -85,B 0,C 180,E1 -11664.477,E2 -11664.477} C_VEL
LIN {X 0,Y 500.933,Z 366.363,A -85,B 0,C 180,E1 -11665.189,E2 -11665.189} C_VEL
LIN {X 0,Y 499.417,Z 363.014,A -85,B 0,C 180,E1 -11665.903,E2 -11665.903} C_VEL
LIN {X 0,Y 497.934,Z 359.493,A -85,B 0,C 180,E1 -11666.653,E2 -11666.653} C_VEL
LIN {X 0,Y 497.913,Z 359.2,A -85,B 0,C 180,E1 -11666.892,E2 -11666.892} C_VEL
LIN {X 0,Y 497.87,Z 359.203,A -85,B 0,C 180,E1 -11670.26,E2 -11670.26} C_VEL
LIN {X 0,Y 497.897,Z 359.191,A -85,B 0,C 180,E1 -11673.652,E2 -11673.652} C_VEL
LIN {X 0,Y 497.914,Z 359.181,A -85,B 0,C 180,E1 -11677.071,E2 -11677.071} C_VEL
LIN {X 0,Y 497.868,Z 359.19,A -85,B 0,C 180,E1 -11680.403,E2 -11680.403} C_VEL
LIN {X 0,Y 497.892,Z 359.206,A -85,B 0,C 180,E1 -11683.91,E2 -11683.91} C_VEL
LIN {X 0,Y 497.913,Z 359.2,A -85,B 0,C 180,E1 -11687.238,E2 -11687.238} C_VEL
LIN {X 0,Y 497.868,Z 359.182,A -85,B 0,C 180,E1 -11690.638,E2 -11690.638} C_VEL
LIN {X 0,Y 497.889,Z 359.199,A -85,B 0,C 180,E1 -11694.121,E2 -11694.121} C_VEL
LIN {X 0,Y 497.923,Z 359.202,A -85,B 0,C 180,E1 -11697.583,E2 -11697.583} C_VEL
LIN {X 0,Y 497.871,Z 359.179,A -85,B 0,C 180,E1 -11700.921,E2 -11700.921} C_VEL
LIN {X 0,Y 497.877,Z 359.202,A -85,B 0,C 180,E1 -11704.492,E2 -11704.492} C_VEL
LIN {X 0,Y 497.925,Z 359.201,A -85,B 0,C 180,E1 -11707.965,E2 -11707.965} C_VEL
LIN {X 0,Y 497.896,Z 359.177,A -85,B 0,C 180,E1 -11711.474,E2 -11711.474} C_VEL
LIN {X 0,Y 497.872,Z 359.2,A -85,B 0,C 180,E1 -11714.896,E2 -11714.896} C_VEL
LIN {X 0,Y 497.905,Z 359.211,A -85,B 0,C 180,E1 -11718.378,E2 -11718.378} C_VEL
LIN {X 0,Y 497.915,Z 359.186,A -85,B 0,C 180,E1 -11721.809,E2 -11721.809} C_VEL
LIN {X 0,Y 497.873,Z 359.185,A -85,B 0,C 180,E1 -11725.199,E2 -11725.199} C_VEL
LIN {X 0,Y 497.894,Z 359.192,A -85,B 0,C 180,E1 -11728.684,E2 -11728.684} C_VEL
LIN {X 0,Y 497.924,Z 359.199,A -85,B 0,C 180,E1 -11732.067,E2 -11732.067} C_VEL
LIN {X 0,Y 497.882,Z 359.207,A -85,B 0,C 180,E1 -11735.575,E2 -11735.575} C_VEL
LIN {X 0,Y 497.896,Z 359.299,A -85,B 0,C 180,E1 -11736.998,E2 -11736.998} C_VEL
LIN {X 0,Y 498.968,Z 362.349,A -85,B 0,C 180,E1 -11737.242,E2 -11737.242} C_VEL
LIN {X 0,Y 501.378,Z 364.864,A -85,B 0,C 180,E1 -11737.68,E2 -11737.68} C_VEL
LIN {X 0,Y 502.405,Z 365.757,A -85,B 0,C 180,E1 -11737.86,E2 -11737.86} C_VEL
LIN {X 0,Y 504.947,Z 369.663,A -85,B 0,C 180,E1 -11738.338,E2 -11738.338} C_VEL
LIN {X 0,Y 506.932,Z 371.815,A -85,B 0,C 180,E1 -11738.684,E2 -11738.684} C_VEL
LIN {X 0,Y 510.263,Z 376.116,A -85,B 0,C 180,E1 -11739.267,E2 -11739.267} C_VEL
LIN {X 0,Y 522.858,Z 392.793,A -85,B 0,C 180,E1 -11741.355,E2 -11741.355} C_VEL
LIN {X 0,Y 535.731,Z 410.892,A -85,B 0,C 180,E1 -11743.325,E2 -11743.325} C_VEL
LIN {X 0,Y 547.57,Z 429.878,A -85,B 0,C 180,E1 -11745.04,E2 -11745.04} C_VEL
LIN {X 0,Y 552.134,Z 438.039,A -85,B 0,C 180,E1 -11745.683,E2 -11745.683} C_VEL
LIN {X 0,Y 543.849,Z 683.906,A -85,B 0,C 180,E1 -11749.233,E2 -11749.233} C_VEL
LIN {X 0,Y 541.705,Z 744.204,A -85,B 0,C 180,E1 -11750.126,E2 -11750.126} C_VEL
LIN {X 0,Y 539.965,Z 768.829,A -85,B 0,C 180,E1 -11750.663,E2 -11750.663} C_VEL
LIN {X 0,Y 537.932,Z 790.735,A -85,B 0,C 180,E1 -11751.296,E2 -11751.296} C_VEL
LIN {X 0,Y 535.138,Z 815.103,A -85,B 0,C 180,E1 -11752.204,E2 -11752.204} C_VEL
LIN {X 0,Y 532.371,Z 835.618,A -85,B 0,C 180,E1 -11753.141,E2 -11753.141} C_VEL
LIN {X 0,Y 528.869,Z 858.448,A -85,B 0,C 180,E1 -11754.387,E2 -11754.387} C_VEL
LIN {X 0,Y 525.676,Z 877.197,A -85,B 0,C 180,E1 -11755.603,E2 -11755.603} C_VEL
LIN {X 0,Y 523.292,Z 890.316,A -85,B 0,C 180,E1 -11756.56,E2 -11756.56} C_VEL
LIN {X 0,Y 521.282,Z 896.832,A -85,B 0,C 180,E1 -11756.997,E2 -11756.997} C_VEL
LIN {X 0,Y 512.667,Z 913.711,A -85,B 0,C 180,E1 -11758.051,E2 -11758.051} C_VEL
LIN {X 0,Y 510.97,Z 918.726,A -85,B 0,C 180,E1 -11758.484,E2 -11758.484} C_VEL
LIN {X 0,Y 507.086,Z 937.373,A -85,B 0,C 180,E1 -11760.41,E2 -11760.41} C_VEL
LIN {X 0,Y 503.657,Z 953.259,A -85,B 0,C 180,E1 -11762.319,E2 -11762.319} C_VEL
LIN {X 0,Y 500.357,Z 968.747,A -85,B 0,C 180,E1 -11764.428,E2 -11764.428} C_VEL
LIN {X 0,Y 497.255,Z 983.636,A -85,B 0,C 180,E1 -11766.789,E2 -11766.789} C_VEL
LIN {X 0,Y 494.795,Z 996.031,A -85,B 0,C 180,E1 -11769.042,E2 -11769.042} C_VEL
LIN {X 0,Y 492.447,Z 1008.915,A -85,B 0,C 180,E1 -11771.779,E2 -11771.779} C_VEL
LIN {X 0,Y 490.905,Z 1018.463,A -85,B 0,C 180,E1 -11774.161,E2 -11774.161} C_VEL
LIN {X 0,Y 489.579,Z 1028.107,A -85,B 0,C 180,E1 -11777.017,E2 -11777.017} C_VEL
LIN {X 0,Y 488.821,Z 1034.962,A -85,B 0,C 180,E1 -11779.511,E2 -11779.511} C_VEL
LIN {X 0,Y 488.319,Z 1041.057,A -85,B 0,C 180,E1 -11782.233,E2 -11782.233} C_VEL
LIN {X 0,Y 488.052,Z 1045.64,A -85,B 0,C 180,E1 -11785.064,E2 -11785.064} C_VEL
LIN {X 0,Y 487.969,Z 1048.417,A -85,B 0,C 180,E1 -11787.534,E2 -11787.534} C_VEL
LIN {X 0,Y 487.93,Z 1050.187,A -85,B 0,C 180,E1 -11790.47,E2 -11790.47} C_VEL
LIN {X 0,Y 487.928,Z 1050.326,A -85,B 0,C 180,E1 -11792.937,E2 -11792.937} C_VEL
LIN {X 0,Y 487.948,Z 1049.337,A -85,B 0,C 180,E1 -11795.409,E2 -11795.409} C_VEL
LIN {X 0,Y 488.031,Z 1046.594,A -85,B 0,C 180,E1 -11798.364,E2 -11798.364} C_VEL
LIN {X 0,Y 488.194,Z 1042.91,A -85,B 0,C 180,E1 -11800.861,E2 -11800.861} C_VEL
LIN {X 0,Y 488.586,Z 1037.768,A -85,B 0,C 180,E1 -11803.491,E2 -11803.491} C_VEL
LIN {X 0,Y 489.35,Z 1030.375,A -85,B 0,C 180,E1 -11806.378,E2 -11806.378} C_VEL
LIN {X 0,Y 490.397,Z 1022.49,A -85,B 0,C 180,E1 -11808.902,E2 -11808.902} C_VEL
LIN {X 0,Y 492.126,Z 1011.581,A -85,B 0,C 180,E1 -11811.794,E2 -11811.794} C_VEL
LIN {X 0,Y 494.034,Z 1001.182,A -85,B 0,C 180,E1 -11814.132,E2 -11814.132} C_VEL
LIN {X 0,Y 496.796,Z 987.389,A -85,B 0,C 180,E1 -11816.798,E2 -11816.798} C_VEL
